REGION Network 17: PU1 Сервис
   IF #Ack OR #PU1.ack.%X3 THEN
       #errServicePU1 := FALSE;   // RS flip-flop
   END_IF;
   IF #PU1.service THEN #errServicePU1 := TRUE; END_IF;
   #PU1.st.%X3 := #errServicePU1;
END_REGION

REGION Network 18: PU2 Сервис
   IF #Ack OR #PU2.ack.%X3 THEN
       #errServicePU2 := FALSE;   // RS flip-flop
   END_IF;
   IF #PU2.service THEN #errServicePU2 := TRUE; END_IF;
   #PU2.st.%X3 := #errServicePU2;
END_REGION

REGION Network 19: Сборная ошибка РU1
   #PU1.error := #errAlarmFC_PU1 OR #errBlock_PU1 OR #errOff_KM_PU1 OR #errOn_KM_PU1 OR #errOff_UZ_PU1 OR #errON_UZ_PU1 OR #errServicePU1;
   #PU1.st.%X10 := #PU1.error;
END_REGION

REGION Network 20: Сборная ошибка РU2
   #PU2.error := #errAlarmFC_PU2 OR #errBlock_PU2 OR #errOff_KM_PU2 OR #errOn_KM_PU2 OR #errOff_UZ_PU1 OR #errON_UZ_PU1 OR #errServicePU2;
   #PU2.st.%X10 := #PU2.error;
END_REGION

REGION Network 21: Состояние работает PU1
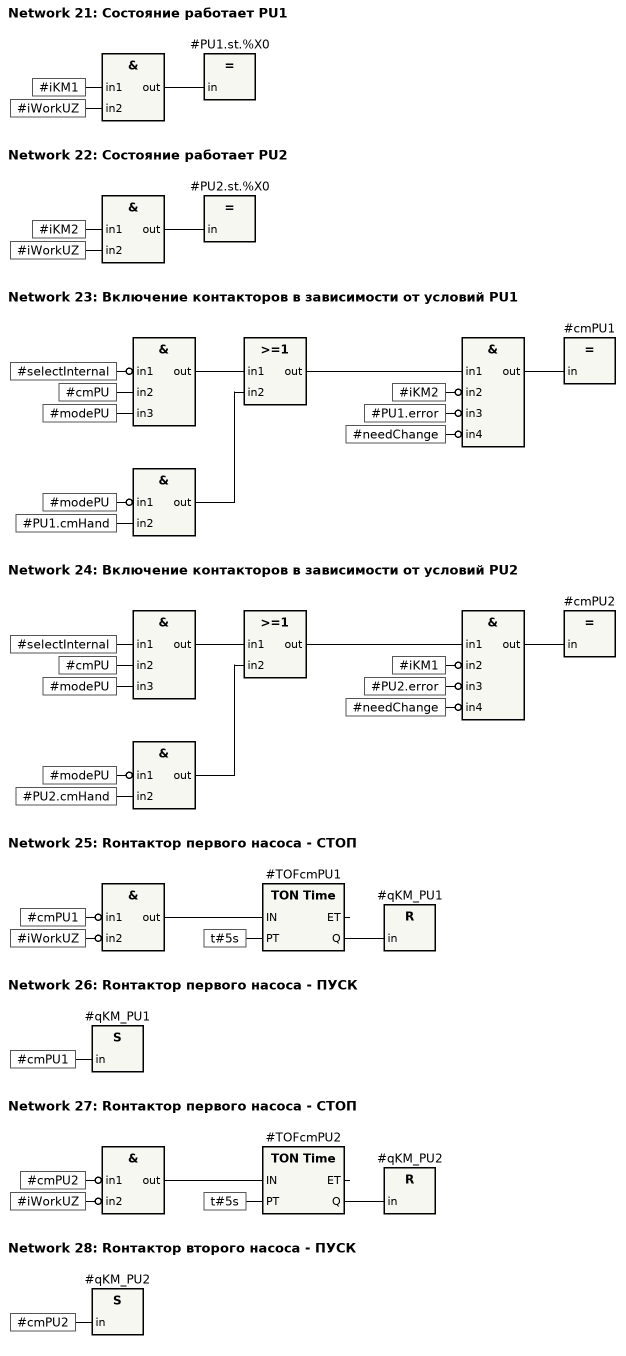
   #PU1.st.%X0 := #iKM1 AND #iWorkUZ;
END_REGION

REGION Network 22: Состояние работает PU2
   #PU2.st.%X0 := #iKM2 AND #iWorkUZ;
END_REGION

REGION Network 23: Включение контакторов в зависимости от условий PU1
   #cmPU1 := ((NOT #selectInternal AND #cmPU AND #modePU) OR (NOT #modePU AND #PU1.cmHand)) AND NOT #iKM2 AND NOT #PU1.error AND NOT #needChange;
END_REGION

REGION Network 24: Включение контакторов в зависимости от условий PU2
   #cmPU2 := ((#selectInternal AND #cmPU AND #modePU) OR (NOT #modePU AND #PU2.cmHand)) AND NOT #iKM1 AND NOT #PU2.error AND NOT #needChange;
END_REGION

REGION Network 25: Rонтактор первого насоса - СТОП
   #TOFcmPU1(IN := NOT #cmPU1 AND NOT #iWorkUZ, PT := t#5s);   // TON
   IF #TOFcmPU1.Q THEN #qKM_PU1 := FALSE; END_IF;
END_REGION

REGION Network 26: Rонтактор первого насоса - ПУСК
   IF #cmPU1 THEN #qKM_PU1 := TRUE; END_IF;
END_REGION

REGION Network 27: Rонтактор первого насоса - СТОП
   #TOFcmPU2(IN := NOT #cmPU2 AND NOT #iWorkUZ, PT := t#5s);   // TON
   IF #TOFcmPU2.Q THEN #qKM_PU2 := FALSE; END_IF;
END_REGION

REGION Network 28: Rонтактор второго насоса - ПУСК
   IF #cmPU2 THEN #qKM_PU2 := TRUE; END_IF;
END_REGION

REGION Network 29: Команда на UZ
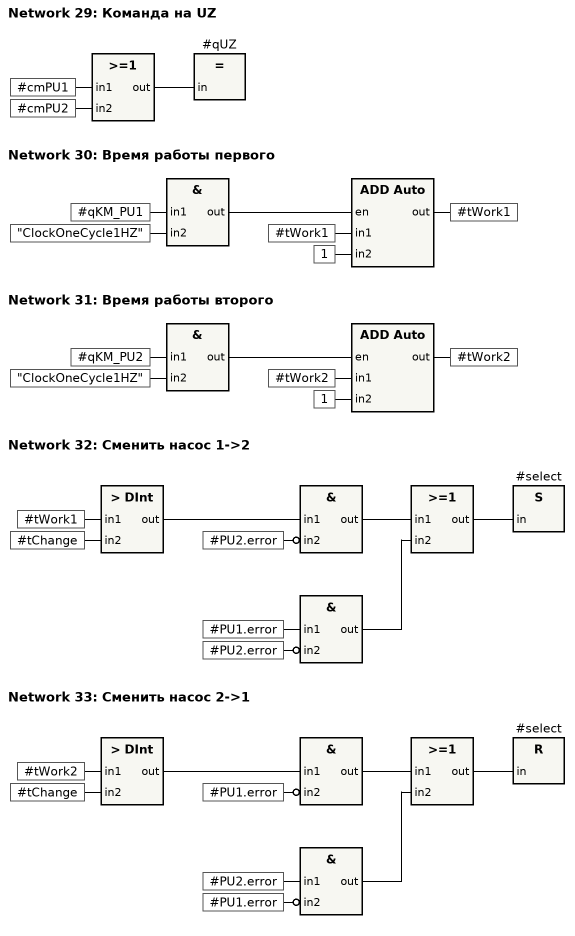
   #qUZ := #cmPU1 OR #cmPU2;
END_REGION

REGION Network 30: Время работы первого
   IF #qKM_PU1 AND "ClockOneCycle1HZ" THEN #tWork1 := #tWork1 + 1; END_IF;
END_REGION

REGION Network 31: Время работы второго
   IF #qKM_PU2 AND "ClockOneCycle1HZ" THEN #tWork2 := #tWork2 + 1; END_IF;
END_REGION

REGION Network 32: Сменить насос 1->2
   IF ((#tWork1 > #tChange) AND NOT #PU2.error) OR (#PU1.error AND NOT #PU2.error) THEN
       #select := TRUE;
   END_IF;
END_REGION

REGION Network 33: Сменить насос 2->1
   IF ((#tWork2 > #tChange) AND NOT #PU1.error) OR (#PU2.error AND NOT #PU1.error) THEN
       #select := FALSE;
   END_IF;
END_REGION

REGION Network 34
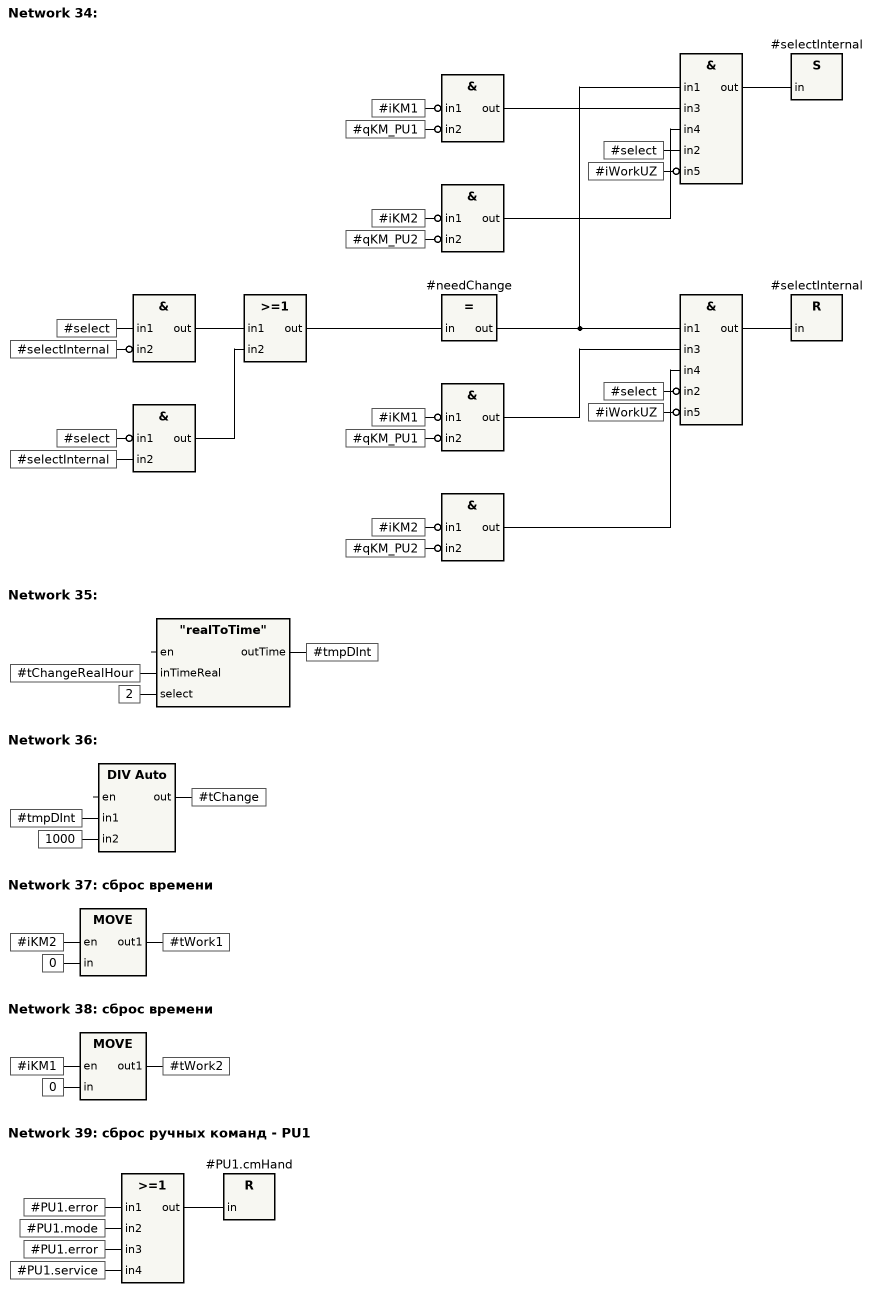
   #needChange := (#select AND NOT #selectInternal) OR (NOT #select AND #selectInternal);
   IF #needChange AND NOT #iKM1 AND NOT #qKM_PU1 AND NOT #iKM2 AND NOT #qKM_PU2 AND #select AND NOT #iWorkUZ THEN
       #selectInternal := TRUE;
   END_IF;
   IF #needChange AND NOT #iKM1 AND NOT #qKM_PU1 AND NOT #iKM2 AND NOT #qKM_PU2 AND NOT #select AND NOT #iWorkUZ THEN
       #selectInternal := FALSE;
   END_IF;
END_REGION

REGION Network 35
   "realToTime"(inTimeReal := #tChangeRealHour, select := 2, outTime => #tmpDInt);
END_REGION

REGION Network 36
   #tChange := #tmpDInt / 1000;
END_REGION

REGION Network 37: сброс времени
   IF #iKM2 THEN #tWork1 := 0; END_IF;
END_REGION

REGION Network 38: сброс времени
   IF #iKM1 THEN #tWork2 := 0; END_IF;
END_REGION

REGION Network 39: сброс ручных команд - PU1
   IF #PU1.error OR #PU1.mode OR #PU1.error OR #PU1.service THEN #PU1.cmHand := FALSE; END_IF;
END_REGION

REGION Network 40: ручная команда - PU2
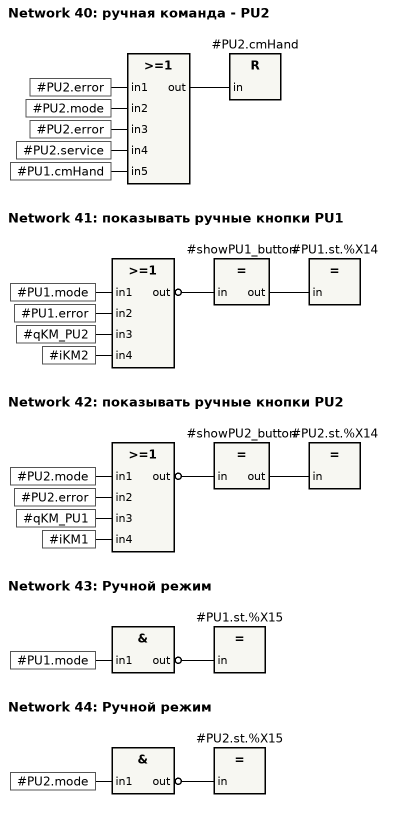
   IF #PU2.error OR #PU2.mode OR #PU2.error OR #PU2.service OR #PU1.cmHand THEN #PU2.cmHand := FALSE; END_IF;
END_REGION

REGION Network 41: показывать ручные кнопки PU1
   #showPU1_button := NOT (#PU1.mode OR #PU1.error OR #qKM_PU2 OR #iKM2);
   #PU1.st.%X14 := #showPU1_button;
END_REGION

REGION Network 42: показывать ручные кнопки PU2
   #showPU2_button := NOT (#PU2.mode OR #PU2.error OR #qKM_PU1 OR #iKM1);
   #PU2.st.%X14 := #showPU2_button;
END_REGION

REGION Network 43: Ручной режим
   #PU1.st.%X15 := NOT #PU1.mode;
END_REGION

REGION Network 44: Ручной режим
   #PU2.st.%X15 := NOT #PU2.mode;
END_REGION

REGION Network 45 (SCL): Сброс битов Ack
   IF NOT #PU1.st.%X0 AND #PU1.ack.%X0 THEN
       #PU1.ack.%X0 := 0;
   END_IF;
   IF NOT #PU1.st.%X1 AND #PU1.ack.%X1 THEN
       #PU1.ack.%X1 := 0;
   END_IF;
   IF NOT #PU1.st.%X2 AND #PU1.ack.%X2 THEN
       #PU1.ack.%X2 := 0;
   END_IF;
   IF NOT #PU1.st.%X3 AND #PU1.ack.%X3 THEN
       #PU1.ack.%X3 := 0;
   END_IF;
   IF NOT #PU1.st.%X4 AND #PU1.ack.%X4 THEN
       #PU1.ack.%X4 := 0;
   END_IF;
   IF NOT #PU1.st.%X5 AND #PU1.ack.%X5 THEN
       #PU1.ack.%X5 := 0;
   END_IF;
   IF NOT #PU1.st.%X6 AND #PU1.ack.%X6 THEN
       #PU1.ack.%X6 := 0;
   END_IF;
   IF NOT #PU1.st.%X7 AND #PU1.ack.%X7 THEN
       #PU1.ack.%X7 := 0;
   END_IF;
   IF NOT #PU1.st.%X8 AND #PU1.ack.%X8 THEN
       #PU1.ack.%X8 := 0;
   END_IF;
   IF NOT #PU1.st.%X9 AND #PU1.ack.%X9 THEN
       #PU1.ack.%X9 := 0;
   END_IF;
   IF NOT #PU1.st.%X10 AND #PU1.ack.%X10 THEN
       #PU1.ack.%X10 := 0;
   END_IF;
   IF NOT #PU1.st.%X11 AND #PU1.ack.%X11 THEN
       #PU1.ack.%X11 := 0;
   END_IF;
   IF NOT #PU1.st.%X12 AND #PU1.ack.%X12 THEN
       #PU1.ack.%X12 := 0;
   END_IF;
   IF NOT #PU1.st.%X13 AND #PU1.ack.%X13 THEN
       #PU1.ack.%X13 := 0;
   END_IF;
   IF NOT #PU1.st.%X14 AND #PU1.ack.%X14 THEN
       #PU1.ack.%X14 := 0;
   END_IF;
   IF NOT #PU1.st.%X15 AND #PU1.ack.%X15 THEN
       #PU1.ack.%X15 := 0;
   END_IF;
   IF NOT #PU2.st.%X0 AND #PU2.ack.%X0 THEN
       #PU2.ack.%X0 := 0;
   END_IF;
   IF NOT #PU2.st.%X1 AND #PU2.ack.%X1 THEN
       #PU2.ack.%X1 := 0;
   END_IF;
   IF NOT #PU2.st.%X2 AND #PU2.ack.%X2 THEN
       #PU2.ack.%X2 := 0;
   END_IF;
   IF NOT #PU2.st.%X3 AND #PU2.ack.%X3 THEN
       #PU2.ack.%X3 := 0;
   END_IF;
   IF NOT #PU2.st.%X4 AND #PU2.ack.%X4 THEN
       #PU2.ack.%X4 := 0;
   END_IF;
   IF NOT #PU2.st.%X5 AND #PU2.ack.%X5 THEN
       #PU2.ack.%X5 := 0;
   END_IF;
   IF NOT #PU2.st.%X6 AND #PU2.ack.%X6 THEN
       #PU2.ack.%X6 := 0;
   END_IF;
   IF NOT #PU2.st.%X7 AND #PU2.ack.%X7 THEN
       #PU2.ack.%X7 := 0;
   END_IF;
   IF NOT #PU2.st.%X8 AND #PU2.ack.%X8 THEN
       #PU2.ack.%X8 := 0;
   END_IF;
   IF NOT #PU2.st.%X9 AND #PU2.ack.%X9 THEN
       #PU2.ack.%X9 := 0;
   END_IF;
   IF NOT #PU2.st.%X10 AND #PU2.ack.%X10 THEN
       #PU2.ack.%X10 := 0;
   END_IF;
   IF NOT #PU2.st.%X11 AND #PU2.ack.%X11 THEN
       #PU2.ack.%X11 := 0;
   END_IF;
   IF NOT #PU2.st.%X12 AND #PU2.ack.%X12 THEN
       #PU2.ack.%X12 := 0;
   END_IF;
   IF NOT #PU2.st.%X13 AND #PU2.ack.%X13 THEN
       #PU2.ack.%X13 := 0;
   END_IF;
   IF NOT #PU2.st.%X14 AND #PU2.ack.%X14 THEN
       #PU2.ack.%X14 := 0;
   END_IF;
   IF NOT #PU2.st.%X15 AND #PU2.ack.%X15 THEN
       #PU2.ack.%X15 := 0;
   END_IF;
END_REGION
END_FUNCTION_BLOCK

FUNCTION "bitToWord" : Void   // FC5, LAD
{ S7_Optimized_Access := 'TRUE' }
VERSION : 0.1
// stored: AutoNumber true, IsIECCheckEnabled false, SetENOAutomatically false, UDAEnableTagReadback false
   VAR_INPUT
      inBit0 : Bool;
      inBit1 : Bool;
      inBit2 : Bool;
      inBit3 : Bool;
      inBit4 : Bool;
      inBit5 : Bool;
      inBit6 : Bool;
      inBit7 : Bool;
      inBit8 : Bool;
      inBit9 : Bool;
      inBit10 : Bool;
      inBit11 : Bool;
      inBit12 : Bool;
      inBit13 : Bool;
      inBit14 : Bool;
      inBit15 : Bool;
   END_VAR
   VAR_OUTPUT
      outWord : Word;
   END_VAR
BEGIN

REGION Network 1
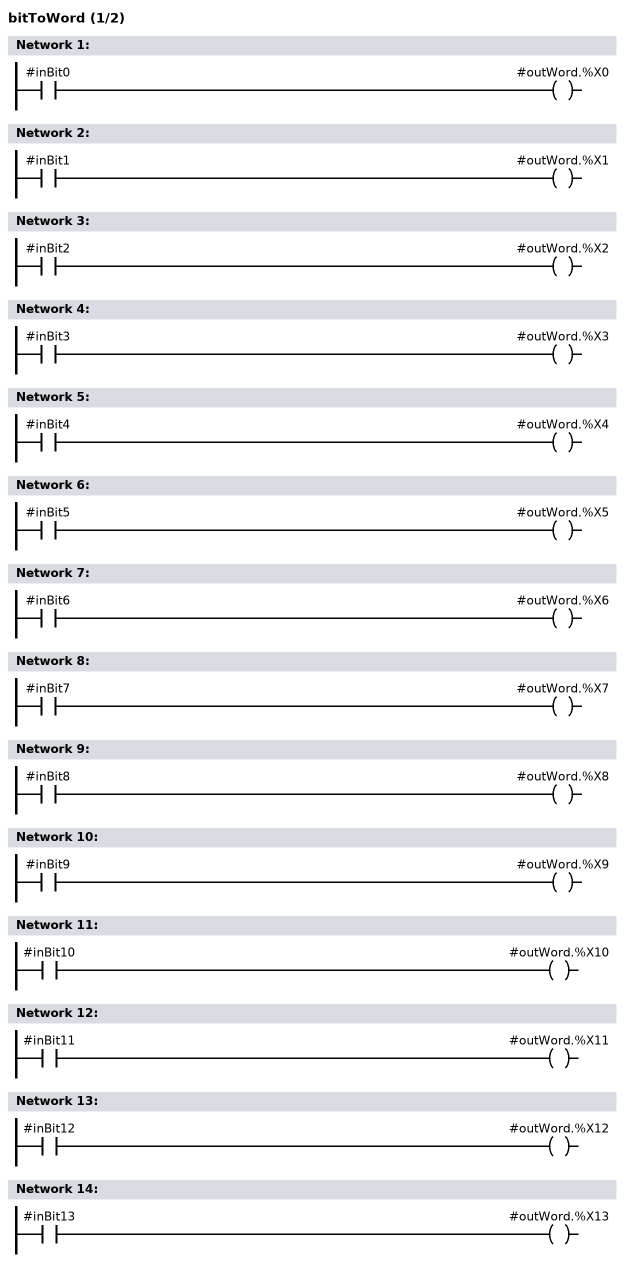
   RUNG wire#powerrail
      Contact( #inBit0 )
      Coil( #outWord.%X0 )
   END_RUNG
   // the same network as SCL:
   #outWord.%X0 := #inBit0;
END_REGION

REGION Network 2
   RUNG wire#powerrail
      Contact( #inBit1 )
      Coil( #outWord.%X1 )
   END_RUNG
   // the same network as SCL:
   #outWord.%X1 := #inBit1;
END_REGION

REGION Network 3
   RUNG wire#powerrail
      Contact( #inBit2 )
      Coil( #outWord.%X2 )
   END_RUNG
   // the same network as SCL:
   #outWord.%X2 := #inBit2;
END_REGION

REGION Network 4
   RUNG wire#powerrail
      Contact( #inBit3 )
      Coil( #outWord.%X3 )
   END_RUNG
   // the same network as SCL:
   #outWord.%X3 := #inBit3;
END_REGION

REGION Network 5
   RUNG wire#powerrail
      Contact( #inBit4 )
      Coil( #outWord.%X4 )
   END_RUNG
   // the same network as SCL:
   #outWord.%X4 := #inBit4;
END_REGION

REGION Network 6
   RUNG wire#powerrail
      Contact( #inBit5 )
      Coil( #outWord.%X5 )
   END_RUNG
   // the same network as SCL:
   #outWord.%X5 := #inBit5;
END_REGION

REGION Network 7
   RUNG wire#powerrail
      Contact( #inBit6 )
      Coil( #outWord.%X6 )
   END_RUNG
   // the same network as SCL:
   #outWord.%X6 := #inBit6;
END_REGION

REGION Network 8
   RUNG wire#powerrail
      Contact( #inBit7 )
      Coil( #outWord.%X7 )
   END_RUNG
   // the same network as SCL:
   #outWord.%X7 := #inBit7;
END_REGION

REGION Network 9
   RUNG wire#powerrail
      Contact( #inBit8 )
      Coil( #outWord.%X8 )
   END_RUNG
   // the same network as SCL:
   #outWord.%X8 := #inBit8;
END_REGION

REGION Network 10
   RUNG wire#powerrail
      Contact( #inBit9 )
      Coil( #outWord.%X9 )
   END_RUNG
   // the same network as SCL:
   #outWord.%X9 := #inBit9;
END_REGION

REGION Network 11
   RUNG wire#powerrail
      Contact( #inBit10 )
      Coil( #outWord.%X10 )
   END_RUNG
   // the same network as SCL:
   #outWord.%X10 := #inBit10;
END_REGION

REGION Network 12
   RUNG wire#powerrail
      Contact( #inBit11 )
      Coil( #outWord.%X11 )
   END_RUNG
   // the same network as SCL:
   #outWord.%X11 := #inBit11;
END_REGION

REGION Network 13
   RUNG wire#powerrail
      Contact( #inBit12 )
      Coil( #outWord.%X12 )
   END_RUNG
   // the same network as SCL:
   #outWord.%X12 := #inBit12;
END_REGION

REGION Network 14
   RUNG wire#powerrail
      Contact( #inBit13 )
      Coil( #outWord.%X13 )
   END_RUNG
   // the same network as SCL:
   #outWord.%X13 := #inBit13;
END_REGION

REGION Network 15
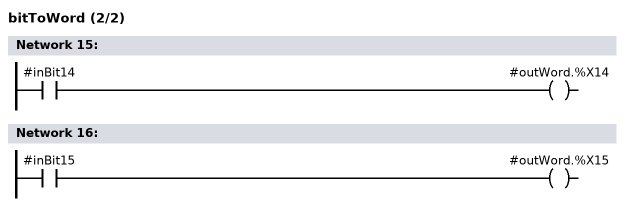
   RUNG wire#powerrail
      Contact( #inBit14 )
      Coil( #outWord.%X14 )
   END_RUNG
   // the same network as SCL:
   #outWord.%X14 := #inBit14;
END_REGION

REGION Network 16
   RUNG wire#powerrail
      Contact( #inBit15 )
      Coil( #outWord.%X15 )
   END_RUNG
   // the same network as SCL:
   #outWord.%X15 := #inBit15;
END_REGION
END_FUNCTION

FUNCTION "VLT_PROFI_FC_BASIC" : Void
TITLE = VLT_PROFI_FC_BASIC
{ S7_Optimized_Access := 'FALSE' }
AUTHOR : Danfoss_Drives
FAMILY : VLT
VERSION : 1.12
//Basic Operation Function Block
   VAR_INPUT 
      sim : Bool;
      ADR : HW_IO;   // S7-1200/1500 requires HW Identifier. Can be found in HW configuration for the specific PPO type
      DRV_EN : Bool;   // Enable Drive. Setting the Drive in Ready to Start mode.
      RUN : Bool;   // Run/Stop drive
      REVERSE : Bool;   // Drive Reverse mode. Also set P4-10 to "both directions" to allow.
      RESET : Bool;   // Reset alarms. Only Trip, not Trip lock.
      REF_VALUE : Real;   // Reference speed 0 - 10000 = 0 - 100.00%
   END_VAR

   VAR_OUTPUT 
      UZ : "UZ_Data";
   END_VAR

   VAR_TEMP 
      PCDRead : Struct   // Pointer to data structure for FC data
         STW : Struct   // Status word
            BIT_00_CTRL_RDY : Bool;   // 0=Control not ready, 1=Control ready
            BIT_01_DRV_RDY : Bool;   // 0=Frequency converter, 1=Frequency converter ready
            BIT_02_COAST_RDY : Bool;   // 0=Coasting, 1=Enable
            BIT_03_TRIP : Bool;   // 0=No error, 1=Trip
            BIT_04_ERROR : Bool;   // 0=No error, 1=Error (no trip)
            BIT_05_RESERVED : Bool;   // 0=Reserved, 1=---
            BIT_06_TRIPLOCK : Bool;   // 0=No error, 1=Triplock
            BIT_07_WARNING : Bool;   // 0=No warning, 1=Warning
            BIT_08_RUNNING_REF : Bool;   // 0=Speed <> reference, 1=Speed=reference
            BIT_09_CTRL_SOURCE : Bool;   // 0=Local operation, 1=Bus control
            BIT_10_F_LIMIT_OK : Bool;   // 0=Out of frequency limit, 1=Frequency limit ok
            BIT_11_IN_OPR : Bool;   // 0=No operation, 1=In operation
            BIT_12_IN_AUTOSTART : Bool;   // 0=Frequency converter OK, 1=Stopped, autostart
            BIT_13_VOLT_MAX : Bool;   // 0=Voltage OK, 1=Voltage exceeded
            BIT_14_TORQ_MAX : Bool;   // 0=Torque OK, 1=Torque exceeded
            BIT_15_TIMER_EXD : Bool;   // 0=Timer OK, 1=Timer exceeded
         END_STRUCT;
         MAV : Int;   // Main actual value
         PCD_02 : Int;   // PCD 02
         PCD_03 : Int;   // PCD 03
         PCD_04 : Int;   // PCD 04
         PCD_05 : Int;   // PCD 05
      END_STRUCT;
      PCDWrite : Struct   // Pointer to data structure for FC data
         CTW : Struct   // Control word
            BIT_00_PRESET_REF_1 : Bool;   // 0=Reference value, 1=selection lsb
            BIT_01_PRESET_REF_2 : Bool;   // 0=Reference value, 1=selection msb
            BIT_02_DC_BRAKE_RAMP : Bool;   // 0=DC brake, 1=Ramp
            BIT_03_COAST_INV : Bool;   // 0=Coasting, 1=No coasting
            BIT_04_QSTP_RMP : Bool;   // 0=Quick stop, 1=Ramp
            BIT_05_HLD_RMP : Bool;   // 0=Hold output frequency, 1=Use ramp
            BIT_06_START : Bool;   // 0=Ramp stop, 1=Start
            BIT_07_RESET : Bool;   // 0=No function, 1=Reset
            BIT_08_JOG : Bool;   // 0=No function, 1=Jog
            BIT_09_RAMP_1_2 : Bool;   // 0=Ramp 1, 1=Ramp 2
            BIT_10_DATA_VALID : Bool;   // 0=Dont use CTW, 1= Use CTW
            BIT_11_RLY_1_ON : Bool;   // 0=Relay 01 deactived, 1=Relay 01 active
            BIT_12_RLY_2_ON : Bool;   // 0=Relay 02 deactived, 1=Relay 02 active
            BIT_13_SETUP_SEL_1 : Bool;   // 0=Parameter set-up, 1=selection lsb
            BIT_14_SETUP_SEL_2 : Bool;   // 0=Parameter set-up, 1=selection msb
            BIT_15_REVERSE : Bool;   // 0= No Reverse, 1= Reverse
         END_STRUCT;
         MRV : Int;   // Main reference value
         PCD_02 : Int;   // PCD 02
         PCD_03 : Int;   // PCD 03
         PCD_04 : Int;   // PCD 04
         PCD_05 : Int;   // PCD 05
      END_STRUCT;
      RDRaw_Data : Array[0..5] of Int;   // Data Read. PROFINET:PPO6 only, with 4 words /PROFIBUS:PPO2 only, with 6 words
      WRRaw_Data : Array[0..5] of Int;   // Data Write. PROFINET:PPO6 only, with 4 words /PROFIBUS:PPO2 only, with 6 words
      RETVAL : Int;   // Return value for DPRD and DPWR for PNET Comm. 0=no fault
      CalcSlope : Real;   // Slope of Ref. value, to convert 0-10000 into 0- 16384
      CurrentInternal : DWord;   // Internal value for current calculation
      PowerInternal : DWord;
      AlwaysOn : Bool;   // Always on
      AlwaysOff : Bool;   // Always off
   END_VAR


BEGIN
	IF #sim THEN
	    #UZ.Ready := 1;
	    #UZ.Fault := 0;
	    #UZ.Warning := 0;
	    #UZ.ErrorConnection := 0;
	    IF #RUN THEN
	        #UZ.MAV := #REF_VALUE;
	        #UZ.Running := 1;
	    ELSE
	        #UZ.MAV := 0;
	        #UZ.Running := 0;
	    END_IF;
	    
	ELSE
	    
	    //-------------------------------------------------------------------------------------------------------------
	    // VLT_PROFI_FC_BASIC: Rev. V1.12
	    // Valid for S7-1200 and S7-1500 Type CPU's.
	    // Block handles communication with a VLT frequency converter. Either Trough PROFINET OR PROFIBUS.
	    // The FC handles basic needs and extraction of Motor current.
	    // PROFINET PPO type is PPO6 (4 words read/Write). PCD2 and PCD3 must be configured for Motor Current.
	    // PROFIBUS PPO type is PPO2 (6 words read/Write). PCD2 and PCD3 must be configured for Motor Current.
	    // Can be done in HW config of S7, on the Drive LCP or MCT10.
	    //-------------------------------------------------------------------------------------------------------------
	    
	    //------------------------------------Standard - Control bits--------------------------------------------------
	    //Can be used locally in Block.
	    #AlwaysOff := false;
	    #AlwaysOn := TRUE;
	    //------------------------------------Standard - Control bits--------------------------------------------------
	    
	    //------------------------------------Read data from fieldbus--------------------------------------------------
	    // Actual data size that is read depends on the Array size.
	    // Minimum size is 4 words.
	    // PPO type can be larger but only the 4 first words are read.
	    // Return value for DPRD and DPWR for PNET Comm. 0=No fault.
	    #RETVAL := DPRD_DAT(LADDR := #ADR, RECORD => #RDRaw_Data);  // Read Raw Data 
	    #UZ.comErr := #RETVAL;
	    //------------------------------------Read data from fieldbus--------------------------------------------------
	    
	    //------------------------------------Read Raw Data is mapped with PCDRead------------------------------------------------------
	    #PCDRead.STW.BIT_00_CTRL_RDY := #RDRaw_Data[0].%X0;
	    #PCDRead.STW.BIT_01_DRV_RDY := #RDRaw_Data[0].%X1;
	    #PCDRead.STW.BIT_02_COAST_RDY := #RDRaw_Data[0].%X2;
	    #PCDRead.STW.BIT_03_TRIP := #RDRaw_Data[0].%X3;
	    #PCDRead.STW.BIT_04_ERROR := #RDRaw_Data[0].%X4;
	    #PCDRead.STW.BIT_05_RESERVED := #RDRaw_Data[0].%X5;
	    #PCDRead.STW.BIT_06_TRIPLOCK := #RDRaw_Data[0].%X6;
	    #PCDRead.STW.BIT_07_WARNING := #RDRaw_Data[0].%X7;
	    #PCDRead.STW.BIT_08_RUNNING_REF := #RDRaw_Data[0].%X8;
	    #PCDRead.STW.BIT_09_CTRL_SOURCE := #RDRaw_Data[0].%X9;
	    #PCDRead.STW.BIT_10_F_LIMIT_OK := #RDRaw_Data[0].%X10;
	    #PCDRead.STW.BIT_11_IN_OPR := #RDRaw_Data[0].%X11;
	    #PCDRead.STW.BIT_12_IN_AUTOSTART := #RDRaw_Data[0].%X12;
	    #PCDRead.STW.BIT_13_VOLT_MAX := #RDRaw_Data[0].%X13;
	    #PCDRead.STW.BIT_14_TORQ_MAX := #RDRaw_Data[0].%X14;
	    #PCDRead.STW.BIT_15_TIMER_EXD := #RDRaw_Data[0].%X15;
	    
	    #PCDRead.MAV := #RDRaw_Data[1];
	    #PCDRead.PCD_02 := #RDRaw_Data[2];
	    #PCDRead.PCD_03 := #RDRaw_Data[3];
	    #PCDRead.PCD_04 := #RDRaw_Data[4];
	    #PCDRead.PCD_05 := #RDRaw_Data[5];
	    //------------------------------------Read Raw Data is mapped with PCDRead------------------------------------------------------
	    
	    //------------------------------------Extraction of Main actual value--------------------------------------------
	    // Main Actual Value(MAV) is read from the Drive as 0 - 16384. Must be converted into 0 - 10000 (0.0 - 100.0 %)
	    IF #UZ.comErr = 0 THEN
	        #CalcSlope := LREAL_TO_REAL(10000.0 / 16384.0);
	        #UZ.MAV := INT_TO_REAL(#PCDRead.MAV) / 163.84; // Convert to percentage (0.0 - 100.0)
	    END_IF;
	    //------------------------------------Extraction of Main actual value--------------------------------------------
	    
	    //------------------------------------Calculation of motor current----------------------------------------------
	    // Motor current is a 32 bit value hence 2 words read from the Drive need to be combined into a DWORD.
	    // Motor current is scaled with 2 decimal points (conversion index -2) hence division by 100.
	    IF #UZ.comErr = 0 THEN
	        #CurrentInternal := DINT_TO_DWORD(#PCDRead.PCD_02); // PCD02 is high word of Motor current
	        #CurrentInternal := SHL_DWORD(IN := #CurrentInternal, N := 16); // Shift high word of Motor current 16 bits to the left
	        #CurrentInternal := #CurrentInternal + DINT_TO_DWORD(#PCDRead.PCD_03); // PCD03 is low word of Motor current
	        #UZ.MotorCurrent := DINT_TO_REAL(DWORD_TO_DINT(#CurrentInternal)) / 100.0;
	        
	        #PowerInternal := DINT_TO_DWORD(#PCDRead.PCD_04);
	        #PowerInternal := SHL_DWORD(IN := #PowerInternal, N := 16);
	        #PowerInternal := #PowerInternal + DINT_TO_DWORD(#PCDRead.PCD_05);
	        #UZ.MotorPower := DINT_TO_REAL(DWORD_TO_DINT(#PowerInternal)) / 100.0;
	    END_IF;
	    //------------------------------------Calculation of Motor current----------------------------------------------
	    
	    //------------------------------------Mask out Drive status bit's-----------------------------------------------
	    IF #UZ.comErr = 0 THEN
	        #UZ.Ready := (#PCDRead.STW.BIT_00_CTRL_RDY AND #PCDRead.STW.BIT_01_DRV_RDY AND #PCDRead.STW.BIT_02_COAST_RDY AND #PCDRead.STW.BIT_09_CTRL_SOURCE); // Drive ready to start from Fieldbus
	        #UZ.Running := #PCDRead.STW.BIT_11_IN_OPR; // Drive is started but not necessarily running on reference speed.
	        #UZ.Run_On_ref := #PCDRead.STW.BIT_08_RUNNING_REF; // Running on reference
	        #UZ.Warning := #PCDRead.STW.BIT_07_WARNING; // Warning present
	        #UZ.Fault := (#PCDRead.STW.BIT_04_ERROR OR #PCDRead.STW.BIT_03_TRIP OR #PCDRead.STW.BIT_06_TRIPLOCK); // Fault present. Trip or Trip lock
	    ELSE
	        #UZ.Ready := FALSE;
	        #UZ.Fault := TRUE;
	    END_IF;
	    //------------------------------------Mask out Drive status bit's-----------------------------------------------
	    
	    //------------------------------------Default settings of Controlword-------------------------------------------
	    // Prepare all Controlword Bit's to default values so that
	    // they are in a "ready to start" mode. CTW =043Ch
	    #PCDWrite.CTW.BIT_00_PRESET_REF_1 := FALSE;
	    #PCDWrite.CTW.BIT_01_PRESET_REF_2 := FALSE;
	    
	    IF #DRV_EN THEN
	        #PCDWrite.CTW.BIT_02_DC_BRAKE_RAMP := TRUE;
	        #PCDWrite.CTW.BIT_03_COAST_INV := TRUE;
	        #PCDWrite.CTW.BIT_04_QSTP_RMP := TRUE;
	        #PCDWrite.CTW.BIT_05_HLD_RMP := TRUE;
	    ELSE
	        #PCDWrite.CTW.BIT_02_DC_BRAKE_RAMP := FALSE;
	        #PCDWrite.CTW.BIT_03_COAST_INV := FALSE;
	        #PCDWrite.CTW.BIT_04_QSTP_RMP := FALSE;
	        #PCDWrite.CTW.BIT_05_HLD_RMP := FALSE;
	    END_IF;
	    
	    #PCDWrite.CTW.BIT_06_START := FALSE;
	    #PCDWrite.CTW.BIT_07_RESET := FALSE;
	    #PCDWrite.CTW.BIT_08_JOG := FALSE;
	    #PCDWrite.CTW.BIT_09_RAMP_1_2 := FALSE;
	    #PCDWrite.CTW.BIT_10_DATA_VALID := TRUE;
	    #PCDWrite.CTW.BIT_11_RLY_1_ON := FALSE;
	    #PCDWrite.CTW.BIT_12_RLY_2_ON := FALSE;
	    #PCDWrite.CTW.BIT_13_SETUP_SEL_1 := FALSE;
	    #PCDWrite.CTW.BIT_14_SETUP_SEL_2 := FALSE;
	    #PCDWrite.CTW.BIT_15_REVERSE := FALSE;
	    //------------------------------------Default settings of Controlword-------------------------------------------
	    
	    //------------------------------------Drive control bit's-------------------------------------------------------
	    #PCDWrite.CTW.BIT_06_START := #RUN AND NOT #UZ.Fault; // Start the Drive if there is no pending Fault.
	    #PCDWrite.CTW.BIT_15_REVERSE := #REVERSE; // Set Drive to Reverse Mode. Ensure Par. 4-10 is set to "Both Directions"
	    #PCDWrite.CTW.BIT_07_RESET := #RESET; // Reset pending Fault
	    //------------------------------------Drive control bit's-------------------------------------------------------
	    
	    //------------------------------------Reference value limit check------------------------------------------------
	    // Must be between 0 - 10000. Ensure reference speed is within limits.
	    IF #REF_VALUE >= 100.00 THEN
	        #REF_VALUE := (100.00);
	    END_IF;
	    IF #REF_VALUE < 0.0 THEN
	        #REF_VALUE := 0.0;
	    END_IF;
	    //------------------------------------Reference value limit check------------------------------------------------
	    
	    //------------------------------------PCDWrite is mapped with WriteRaw data--------------------------------------------------
	    #WRRaw_Data[0].%X0 := #PCDWrite.CTW.BIT_00_PRESET_REF_1;
	    #WRRaw_Data[0].%X1 := #PCDWrite.CTW.BIT_01_PRESET_REF_2;
	    #WRRaw_Data[0].%X2 := #PCDWrite.CTW.BIT_02_DC_BRAKE_RAMP;
	    #WRRaw_Data[0].%X3 := #PCDWrite.CTW.BIT_03_COAST_INV;
	    #WRRaw_Data[0].%X4 := #PCDWrite.CTW.BIT_04_QSTP_RMP;
	    #WRRaw_Data[0].%X5 := #PCDWrite.CTW.BIT_05_HLD_RMP;
	    #WRRaw_Data[0].%X6 := #PCDWrite.CTW.BIT_06_START;
	    #WRRaw_Data[0].%X7 := #PCDWrite.CTW.BIT_07_RESET;
	    #WRRaw_Data[0].%X8 := #PCDWrite.CTW.BIT_08_JOG;
	    #WRRaw_Data[0].%X9 := #PCDWrite.CTW.BIT_09_RAMP_1_2;
	    #WRRaw_Data[0].%X10 := #PCDWrite.CTW.BIT_10_DATA_VALID;
	    #WRRaw_Data[0].%X11 := #PCDWrite.CTW.BIT_11_RLY_1_ON;
	    #WRRaw_Data[0].%X12 := #PCDWrite.CTW.BIT_12_RLY_2_ON;
	    #WRRaw_Data[0].%X13 := #PCDWrite.CTW.BIT_13_SETUP_SEL_1;
	    #WRRaw_Data[0].%X14 := #PCDWrite.CTW.BIT_14_SETUP_SEL_2;
	    #WRRaw_Data[0].%X15 := #PCDWrite.CTW.BIT_15_REVERSE;
	    
	    #WRRaw_Data[2] := #PCDWrite.PCD_02;
	    #WRRaw_Data[3] := #PCDWrite.PCD_03;
	    //------------------------------------PCDWrite is mapped with WriteRaw data--------------------------------------------------
	    
	    //------------------------------------Reference value limit check------------------------------------------------
	    // Must be between 0 - 10000. Ensure reference speed is within limits.
	    IF #REF_VALUE >= 100.00 THEN
	        #REF_VALUE := 100.00;
	    END_IF;
	    IF #REF_VALUE < 0.0 THEN
	        #REF_VALUE := 0.0;
	    END_IF;
	    //------------------------------------Reference value limit check------------------------------------------------
	    
	    //------------------------------------Prepare Reference value----------------------------------------------------
	    // PCD Write block position 1. Fit's with PPO type mapping
	    // Convert 10000 into 16384 which equals 4000h. 10000 = 100.00%
	    #CalcSlope := LREAL_TO_REAL(16384.0 / 10000.0);
	    #PCDWrite.MRV := REAL_TO_INT(#REF_VALUE * 163.84);
	    //FLOOR_INT(#CalcSlope * #REF_VALUE); // Convert to percentage (0.0 - 100.0)
	    #WRRaw_Data[1] := #PCDWrite.MRV; // Main reference value is Mapped with write Raw Data
	    //------------------------------------Prepare Reference value----------------------------------------------------
	    
	    //------ADR------------------------------Send Data------------------------------------------------------------------
	    // Return value for DPRD and DPWR for PNET Comm. 0=No fault
	    IF #UZ.comErr = 0 THEN
	        #RETVAL := DPWR_DAT(LADDR := #ADR, RECORD := #WRRaw_Data); //#Write Raw Data);
	        #UZ.comErr := #RETVAL;
	    END_IF;
	    //------------------------------------Send Data------------------------------------------------------------------
	    
	    
	    IF #UZ.comErr = 0 THEN
	        #UZ.ErrorConnection := 0;
	    ELSE
	        #UZ.ErrorConnection := 1;
	    END_IF;
	    
	END_IF;
	
	//------------------------------------Ensure ENO is TRUE always--------------------------------------------------
	ENO := TRUE;
	//------------------------------------Ensure ENO is TRUE always--------------------------------------------------
	
END_FUNCTION

FUNCTION_BLOCK "AllDpump"
{ S7_Optimized_Access := 'TRUE' }
VERSION : 0.1
   VAR 
      dp101 : "DPumpCntr";
      dp501 : "DPumpCntr";
      dp502 : "DPumpCntr";
      dp801 : "DPumpCntr";
      dp802 : "DPumpCntr";
      dp803 : "DPumpCntr";
      dp1001 : "DPumpCntr";
   END_VAR


BEGIN
	
	REGION Dpumps handlers
	    #dp101(power := TRUE,
	           run := "iDP101_Run",
	           emrStop := TRUE,
	           alarmFC := "iDP101_Fail",
	           Ack := "dbMain".Ack,
	           FE := 0.0,
	           qStart => "qDP101_Start",
	           pqw => "aqDP101",
	           dev := "dtDpump".dp101,
	           prop := "dtPropDpump".dp101);
	    
	    #dp501(power := TRUE,
	           run := "iDP501_Run",
	           emrStop := TRUE,
	           alarmFC := "iDP501_Fail",
	           Ack := "dbMain".Ack,
	           FE := 0.0,
	           qStart => "qDP501_Start",
	           pqw => "aqDP501",
	           dev := "dtDpump".dp501,
	           prop := "dtPropDpump".dp501);
	    
	    #dp502(power := TRUE,
	           run := "iDP502_Run",
	           emrStop := TRUE,
	           alarmFC := "iDP502_Fail",
	           Ack := "dbMain".Ack,
	           FE := 0.0,
	           qStart => "qDP502_Start",
	           pqw => "aqDP502",
	           dev := "dtDpump".dp502,
	           prop := "dtPropDpump".dp502);
	    
	    #dp801(power := TRUE,
	           run := "iDP801_Run",
	           emrStop := TRUE,
	           alarmFC := "iDP801_Fail",
	           Ack := "dbMain".Ack,
	           FE := 0.0,
	           qStart => "qDP801_Start",
	           pqw => "aqDP801",
	           dev := "dtDpump".dp801,
	           prop := "dtPropDpump".dp801);
	    
	    #dp802(power := TRUE,
	           run := "iDP802_Run",
	           emrStop := TRUE,
	           alarmFC := "iDP802_Fail",
	           Ack := "dbMain".Ack,
	           FE := 0.0,
	           qStart => "qDP802_Start",
	           pqw => "aqDP802",
	           dev := "dtDpump".dp802,
	           prop := "dtPropDpump".dp802);
	    
	    #dp803(power := TRUE,
	           run := "iDP803_Run",
	           emrStop := TRUE,
	           alarmFC := "iDP803_Fail",
	           Ack := "dbMain".Ack,
	           FE := 0.0,
	           qStart => "qDP803_Start",
	           pqw => "aqDP803",
	           dev := "dtDpump".dp803,
	           prop := "dtPropDpump".dp803);
	    
	    #dp1001(power := TRUE,
	            run := "iDP1001_Run",
	            emrStop := TRUE,
	            alarmFC := "iDP1001_Fail",
	            Ack := "dbMain".Ack,
	            FE := 0.0,
	            qStart => "qDP1001_Start",
	            pqw => "aqDP1001",
	            dev := "dtDpump".dp1001,
	            prop := "dtPropDpump".dp1001);
	END_REGION
	
END_FUNCTION_BLOCK

FUNCTION_BLOCK "DPumpCntr"   // FB70, LAD
{ S7_Optimized_Access := 'FALSE' }
VERSION : 0.1
// #ST:
// номер бита, часло десятичное
//  0  - стоп 
// 0 1 - работа
// 1 2 - запуск
// 2 4 - остановка
// 3 8 - сервисный режим
// 4 16 - ошибка Пуска
// 5 32 - ошибка Стопа
// 6 64 - ошибка питания
// 7 128 - ошибка частотника (дозатора)
// 8 256 - Блокировка внешняя
// 9 - 512 - нажат аварийный стоп
// 10 -1024 - сборная авария
// 11 2048
// 12 4096
// 13 8192
// 14 16384 
// 15 32768 - режим 0-ручной, 1-авто
// 
// 
// 
// показывать кнопки ручного управления
// stored: AutoNumber false, IsIECCheckEnabled false, SetENOAutomatically false, UDAEnableTagReadback false
   VAR_INPUT
      power : Bool;   // питание устройства
      run : Bool;
      emrStop : Bool;   // Авариный стоп 0-авария, 1-ок
      alarmFC : Bool;   // 1-авария
      Ack : Bool;   // Сброс Аварий
      FE : Real;
   END_VAR
   VAR_OUTPUT
      qStart : Bool;
      pqw : Int;
   END_VAR
   VAR_IN_OUT
      dev : "DPump";
      prop : "PropDosing";
   END_VAR
   VAR DB_SPECIFIC
      ErrOC : Bool;   // Признак аварии по закрытию или открытию
      ErrPower : Bool;   // Признак аварии питания
      ErrDis : Bool;   // Признак внешней блокировки
      qON : Bool;   // Выход для управления механизмом
      tmrClosing { S7_SetPoint := 'True'} : TON_TIME;
      tmrOpening { S7_SetPoint := 'True'} : TON_TIME;
      closed : Bool;
      opened : Bool;
      closing : Bool;
      opening : Bool;
      errStart : Bool;
      errStop : Bool;
      errEmrStop : Bool;
      errAlarmFc : Bool;
      errService : Bool;
      tStart : Time;
      tStop : Time;
   END_VAR
   VAR
      ServiceEventHandler { S7_SetPoint := 'True'} : "DevAckSingleAlarm";
      PowerEventHandler { S7_SetPoint := 'True'} : "DevAckSingleAlarm";
      DevAlarmEventHandler { S7_SetPoint := 'True'} : "DevAckSingleAlarm";
      DisEventHandler { S7_SetPoint := 'True'} : "DevAckSingleAlarm";
      EmrStopEventHandler { S7_SetPoint := 'True'} : "DevAckSingleAlarm";
      BadStartEventHandler { S7_SetPoint := 'True'} : "DevAckSingleAlarm";
      BadStopEventHandler { S7_SetPoint := 'True'} : "DevAckSingleAlarm";
   END_VAR
BEGIN

REGION Network 1: Сброс состояния
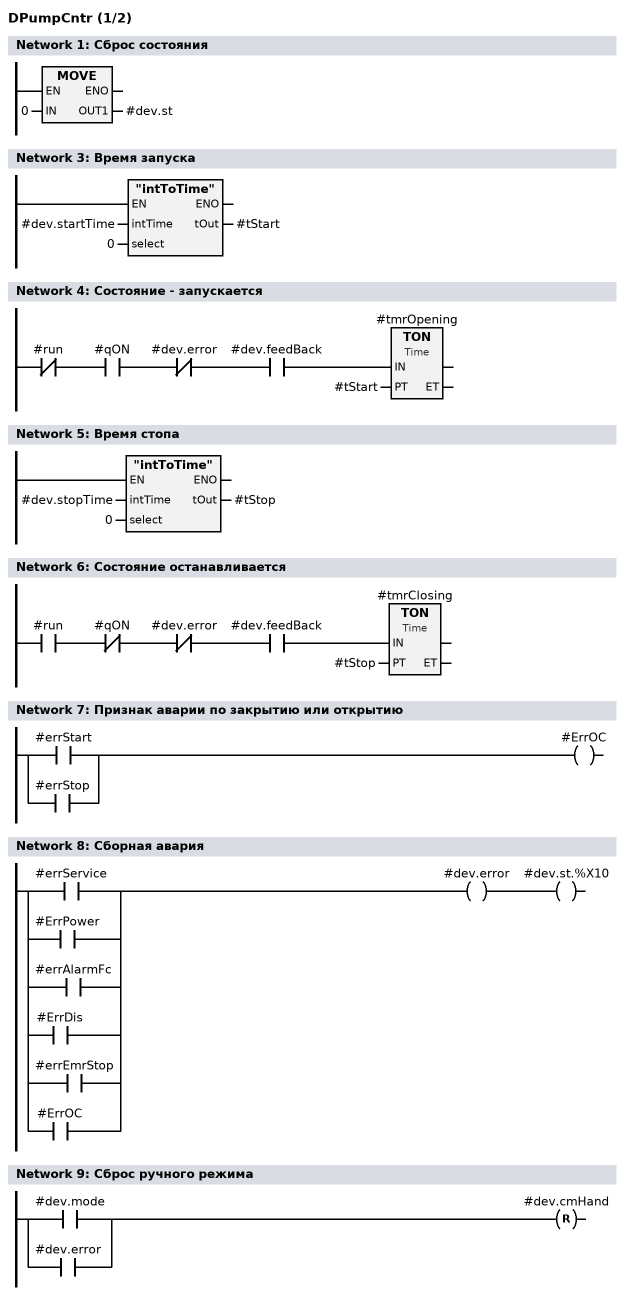
   RUNG wire#powerrail
      { S7_GenerateENO := "TRUE" } Move(in := 0, out1 => #dev.st)
   END_RUNG
   // the same network as SCL:
   #dev.st := 0;
END_REGION

REGION Network 2 (SCL): Event handlers
   #ServiceEventHandler(alarmSignal := #dev.service,
                        ack := #Ack,
                        ackBit := #dev.ack.%X3,
                        stateBit := #dev.st.%X3,
                        alarmTag := #errService);
   #BadStartEventHandler(alarmSignal:=#tmrOpening.Q,
                         ack:=#Ack,
                         ackBit:=#dev.ack.%X4,
                         stateBit:=#dev.st.%X4,
                         alarmTag:=#errStart);
   #BadStopEventHandler(alarmSignal:=#tmrClosing.Q,
                        ack:=#Ack,
                        ackBit:=#dev.ack.%X5,
                        stateBit:=#dev.ack.%X5,
                        alarmTag:=#errStop);
   #PowerEventHandler(alarmSignal := #power,
                      ack := #Ack,
                      ackBit := #dev.ack.%X6,
                      stateBit := #dev.st.%X6,
                      alarmTag := #ErrPower);
   #DevAlarmEventHandler(alarmSignal := #alarmFC,
                         ack := #Ack,
                         ackBit := #dev.ack.%X7,
                         stateBit := #dev.st.%X7,
                         alarmTag := #errAlarmFc);
   #DisEventHandler(alarmSignal := #dev.block,
                    ack := #Ack,
                    ackBit := #dev.ack.%X8,
                    stateBit := #dev.st.%X8,
                    alarmTag := #ErrDis);
   #EmrStopEventHandler(alarmSignal := #emrStop,
                        ack := #Ack,
                        ackBit := #dev.ack.%X9,
                        stateBit := #dev.st.%X9,
                        alarmTag := #errEmrStop);
END_REGION

REGION Network 3: Время запуска
   RUNG wire#powerrail
      "intToTime"(intTime := #dev.startTime, select := 0, tOut => #tStart)
   END_RUNG
   // the same network as SCL:
   "intToTime"(intTime := #dev.startTime, select := 0, tOut => #tStart);
END_REGION

REGION Network 4: Состояние - запускается
   RUNG wire#powerrail
      I_Contact( #run )
      Contact( #qON )
      I_Contact( #dev.error )
      Contact( #dev.feedBack )
      { S7_Templates := "time_type := Time" } #tmrOpening.TON(pt := #tStart, et =>)
   END_RUNG
   // the same network as SCL:
   #tmrOpening(IN := NOT #run AND #qON AND NOT #dev.error AND #dev.feedBack, PT := #tStart);   // TON
END_REGION

REGION Network 5: Время стопа
   RUNG wire#powerrail
      "intToTime"(intTime := #dev.stopTime, select := 0, tOut => #tStop)
   END_RUNG
   // the same network as SCL:
   "intToTime"(intTime := #dev.stopTime, select := 0, tOut => #tStop);
END_REGION

REGION Network 6: Состояние останавливается
   RUNG wire#powerrail
      Contact( #run )
      I_Contact( #qON )
      I_Contact( #dev.error )
      Contact( #dev.feedBack )
      { S7_Templates := "time_type := Time" } #tmrClosing.TON(pt := #tStop, et =>)
   END_RUNG
   // the same network as SCL:
   #tmrClosing(IN := #run AND NOT #qON AND NOT #dev.error AND #dev.feedBack, PT := #tStop);   // TON
END_REGION

REGION Network 7: Признак аварии по закрытию или открытию
   RUNG wire#powerrail
      Contact( #errStart )
      wire#w1
      Coil( #ErrOC )
   END_RUNG
   RUNG wire#powerrail
      Contact( #errStop )
   END_RUNG wire#w1
   // the same network as SCL:
   #ErrOC := #errStart OR #errStop;
END_REGION

REGION Network 8: Сборная авария
   RUNG wire#powerrail
      Contact( #errService )
      wire#w1
      Coil( #dev.error )
      Coil( #dev.st.%X10 )
   END_RUNG
   RUNG wire#powerrail
      Contact( #ErrPower )
   END_RUNG wire#w1
   RUNG wire#powerrail
      Contact( #errAlarmFc )
   END_RUNG wire#w1
   RUNG wire#powerrail
      Contact( #ErrDis )
   END_RUNG wire#w1
   RUNG wire#powerrail
      Contact( #errEmrStop )
   END_RUNG wire#w1
   RUNG wire#powerrail
      Contact( #ErrOC )
   END_RUNG wire#w1
   // the same network as SCL:
   #dev.error := #errService OR #ErrPower OR #errAlarmFc OR #ErrDis OR #errEmrStop OR #ErrOC;
   #dev.st.%X10 := #dev.error;
END_REGION

REGION Network 9: Сброс ручного режима
   RUNG wire#powerrail
      Contact( #dev.mode )
      wire#w1
      R_Coil( #dev.cmHand )
   END_RUNG
   RUNG wire#powerrail
      Contact( #dev.error )
   END_RUNG wire#w1
   // the same network as SCL:
   IF #dev.mode OR #dev.error THEN #dev.cmHand := FALSE; END_IF;
END_REGION

REGION Network 10: Сброс авто режима
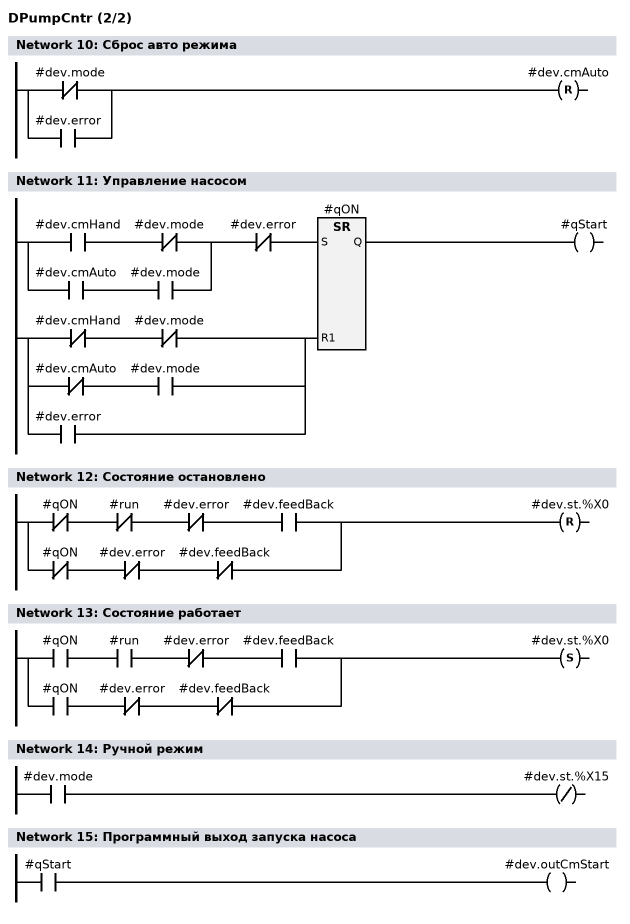
   RUNG wire#powerrail
      I_Contact( #dev.mode )
      wire#w1
      R_Coil( #dev.cmAuto )
   END_RUNG
   RUNG wire#powerrail
      Contact( #dev.error )
   END_RUNG wire#w1
   // the same network as SCL:
   IF NOT #dev.mode OR #dev.error THEN #dev.cmAuto := FALSE; END_IF;
END_REGION

REGION Network 11: Управление насосом
   RUNG wire#powerrail
      Contact( #dev.cmHand )
      I_Contact( #dev.mode )
      wire#w1
      I_Contact( #dev.error )
      S_SR(operand := #qON, r1 := wire#w2)
      Coil( #qStart )
   END_RUNG
   RUNG wire#powerrail
      Contact( #dev.cmAuto )
      Contact( #dev.mode )
   END_RUNG wire#w1
   RUNG wire#powerrail
      I_Contact( #dev.cmHand )
      I_Contact( #dev.mode )
   END_RUNG wire#w2
   RUNG wire#powerrail
      I_Contact( #dev.cmAuto )
      Contact( #dev.mode )
   END_RUNG wire#w2
   RUNG wire#powerrail
      Contact( #dev.error )
   END_RUNG wire#w2
   // the same network as SCL:
   IF ((#dev.cmHand AND NOT #dev.mode) OR (#dev.cmAuto AND #dev.mode)) AND NOT #dev.error THEN
       #qON := TRUE;   // SR flip-flop
   END_IF;
   IF (NOT #dev.cmHand AND NOT #dev.mode) OR (NOT #dev.cmAuto AND #dev.mode) OR #dev.error THEN
       #qON := FALSE;
   END_IF;
   #qStart := #qON;
END_REGION

REGION Network 12: Состояние остановлено
   RUNG wire#powerrail
      I_Contact( #qON )
      I_Contact( #run )
      I_Contact( #dev.error )
      Contact( #dev.feedBack )
      wire#w1
      R_Coil( #dev.st.%X0 )
   END_RUNG
   RUNG wire#powerrail
      I_Contact( #qON )
      I_Contact( #dev.error )
      I_Contact( #dev.feedBack )
   END_RUNG wire#w1
   // the same network as SCL:
   IF (NOT #qON AND NOT #run AND NOT #dev.error AND #dev.feedBack) OR (NOT #qON AND NOT #dev.error AND NOT #dev.feedBack) THEN
       #dev.st.%X0 := FALSE;
   END_IF;
END_REGION

REGION Network 13: Состояние работает
   RUNG wire#powerrail
      Contact( #qON )
      Contact( #run )
      I_Contact( #dev.error )
      Contact( #dev.feedBack )
      wire#w1
      S_Coil( #dev.st.%X0 )
   END_RUNG
   RUNG wire#powerrail
      Contact( #qON )
      I_Contact( #dev.error )
      I_Contact( #dev.feedBack )
   END_RUNG wire#w1
   // the same network as SCL:
   IF (#qON AND #run AND NOT #dev.error AND #dev.feedBack) OR (#qON AND NOT #dev.error AND NOT #dev.feedBack) THEN
       #dev.st.%X0 := TRUE;
   END_IF;
END_REGION

REGION Network 14: Ручной режим
   RUNG wire#powerrail
      Contact( #dev.mode )
      I_Coil( #dev.st.%X15 )
   END_RUNG
   // the same network as SCL:
   #dev.st.%X15 := NOT #dev.mode;
END_REGION

REGION Network 15: Программный выход запуска насоса
   RUNG wire#powerrail
      Contact( #qStart )
      Coil( #dev.outCmStart )
   END_RUNG
   // the same network as SCL:
   #dev.outCmStart := #qStart;
END_REGION

REGION Network 16 (SCL): Prop dossing
   //дозирование пропорционально расходу

   //производителньность л/ч

   IF #dev.mode AND #dev.cmAuto THEN
       //KVA
       IF #prop.enableFix THEN
           IF #prop.fixSP > 100 THEN
               #prop.fixSP := 100;
           END_IF;
           IF #prop.fixSP < 0 THEN
               #prop.fixSP := 0;
           END_IF;
           #prop.outLPH := (#prop.max * #prop.fixSP) / 100;
           //
           // #prop.outLPH := #prop.fixSP;
       ELSE
           IF #prop.density > 0 THEN
               #prop.outLPH := #FE * #prop.spAuto / (#prop.density * 1000.0);
           ELSE
               #prop.outLPH := 0;
           END_IF;

           //запрет дозирования если расход меньше заданного
           IF #FE < #prop.minFE THEN
               #prop.outLPH := 0.0;
           END_IF;
       END_IF;
   END_IF;
   IF NOT #dev.mode AND #dev.cmHand THEN
       #prop.outLPH := #prop.spHand;
   END_IF;

   //запрет дозирования
   IF NOT #dev.cmHand AND NOT #dev.cmAuto THEN
       #prop.outLPH := 0.0;
   END_IF;

   IF #prop.outLPH > #prop.max THEN
       #prop.outLPH := #prop.max;
   END_IF;

   //расчет PQW
   IF #prop.max > 0 THEN
       #pqw := REAL_TO_INT(#prop.outLPH * 27648.0 / #prop.max);
   ELSE
       #pqw := 0;
   END_IF;

   //ограничение выхода
   IF #pqw < 0 THEN
       #pqw := 0;
   END_IF;
   IF #pqw > 27648 THEN
       #pqw := 27648;
   END_IF;
   //расчет тока
   #prop.outmA := 4.0 + INT_TO_REAL(#pqw) * 16.0 / 27648.0;
   #prop.outSP := INT_TO_REAL(#pqw) * 100.0 / 27648.0;
   #prop.FE := #FE;
END_REGION
END_FUNCTION_BLOCK

FUNCTION_BLOCK "AllUF"
{ S7_Optimized_Access := 'TRUE' }
VERSION : 0.1
   VAR 
      reqNumbWorkUF { ExternalVisible := 'False'; ExternalWritable := 'False'} : USInt;
      readyUF : Array[0..1] of Bool;
      workUF : Array[0..1] of Bool;
      cmUF : Array[0..1] of Bool;
      HandlerUF1 : "HandlerUF";
      HandlerUF2 : "HandlerUF";
   END_VAR

   VAR_TEMP 
      tChModeUF1 : Bool;
      tChModeUF2 : Bool;
      tErr : Bool;
   END_VAR

   VAR CONSTANT 
      UF1 : Int := 0;
      UF2 : Int := 1;
   END_VAR


BEGIN
	REGION Device mode for UF12 and UF34
	    //Valves UF1
	    "dtAV".DVA501.mode :=
	    "dtAV".DVA503.mode :=
	    "dtAV".DVA505.mode :=
	    "dtAV".DVA507.mode :=
	    "dtAV".DVA508.mode :=
	    "dtAV".DVA509.mode :=
	    "dtAV".DVA512.mode :=
	    "dtUF".modeUF1;
	    //Valves UF2
	    "dtAV".DVA502.mode :=
	    "dtAV".DVA510.mode :=
	    "dtAV".DVA513.mode :=
	    "dtAV".DVA514.mode :=
	    "dtAV".DVA515.mode :=
	    "dtAV".DVA516.mode :=
	    "dtAV".DVA506.mode :=
	    "dtUF".modeUF2;
	    //Common devices
	    "dtAV".DVA504.mode :=
	    "dtAV".DVA511.mode :=
	    //    "dtPump".P701.mode :=
	    //    "dtPump".P701.mode :=
	    "dtUF".modeUF1 OR "dtUF".modeUF2;
	END_REGION
	REGION Calculate number of UF in work
	    // "CalcNumDevUf"(cmStart:= "dtUF".cmAuto,
	    //                nWorkDev:=#reqNumbWorkUF,
	    //                lev:= "dtAnalogData".et_data["aiLT601"].Par,
	    //                levStop1:="dtParmUF".filtrateStopLevUF1,
	    //                levStart1:="dtParmUF".filtrateStartLevUF1,
	    //                levStop2:="dtParmUF".filtrateStopLevUF2,
	    //                levStart2:="dtParmUF".filtrateStartLevUF2,
	    //                settingsError=>"dtParmUF".errSettingsLev,
	    //                nNeedWork:=#reqNumbWorkUF);
	END_REGION
	REGION Prepare FOR select work UF
	    #readyUF[#UF1] := "dtUF".modeUF1
	    AND NOT (
	    "dtUF".flagUF1.Err OR
	    "dtUF".flagUF1.HW OR
	    "dtUF".flagUF1.HW_A OR
	    "dtUF".flagUF1.CEB1 OR
	    "dtUF".flagUF1.CEB1_A OR
	    "dtUF".flagUF1.CEB2 OR
	    "dtUF".flagUF1.CEB2_A
	    );
	    #readyUF[#UF2] := "dtUF".modeUF2
	    AND NOT (
	    "dtUF".flagUF2.Err OR
	    "dtUF".flagUF2.HW OR
	    "dtUF".flagUF2.HW_A OR
	    "dtUF".flagUF2.CEB1 OR
	    "dtUF".flagUF2.CEB1_A OR
	    "dtUF".flagUF2.CEB2 OR
	    "dtUF".flagUF2.CEB2_A
	    );
	    
	    #workUF[#UF1] := "dtUF".flagUF1.Filtration AND #readyUF[#UF1];
	    #workUF[#UF2] := "dtUF".flagUF2.Filtration AND #readyUF[#UF2];
	END_REGION
	REGION Select work UF
	    "DevInWork"(ReqNumbWorkDev := #reqNumbWorkUF,
	                ReadyDev:=#readyUF,
	                WorkDev := #workUF,
	                DevCm => #cmUF,
	                ErrNotSameBound => #tErr);
	    
	    IF #cmUF[#UF1] AND "dtUF".flagUF1.StandBy THEN
	        #HandlerUF1.cmUF := "UF_CM_START";
	    END_IF;
	    IF NOT (#cmUF[#UF1]) AND "dtUF".flagUF1.Filtration THEN
	        #HandlerUF1.cmUF := "UF_CM_STOP";
	    END_IF;
	    
	    IF #cmUF[#UF2] AND "dtUF".flagUF2.StandBy THEN
	        #HandlerUF2.cmUF := "UF_CM_START";
	    END_IF;
	    IF NOT (#cmUF[#UF2]) AND "dtUF".flagUF2.Filtration THEN
	        #HandlerUF2.cmUF := "UF_CM_STOP";
	    END_IF;
	END_REGION
	REGION Block wash
	    //UF1
	    "dtUF".bUF2.HW :=
	    "dtUF".bUF2.CEB1 :=
	    "dtUF".bUF2.CEB2 :=
	    "dtUF".flagUF2.HW
	    OR "dtUF".flagUF2.HW_A
	    OR "dtUF".flagUF2.CEB1
	    OR "dtUF".flagUF2.CEB1_A
	    OR "dtUF".flagUF2.CEB2
	    OR "dtUF".flagUF2.CEB2_A;
	    
	    "dtUF".bUF2.HW_A :=
	    "dtUF".bUF2.CEB1_A :=
	    "dtUF".bUF2.CEB2_A :=
	    "dtUF".flagUF2.HW
	//    OR ("dtAnalogData".et_data["iwLT601"].Par <= "dtParmUF".minFiltrLevForWash)
	    OR "dtUF".flagUF2.HW_A
	    OR "dtUF".flagUF2.CEB1
	    OR "dtUF".flagUF2.CEB1_A
	    OR "dtUF".flagUF2.CEB2
	    OR "dtUF".flagUF2.CEB2_A;
	
	    //UF2
	    "dtUF".bUF2.HW :=
	    "dtUF".bUF2.CEB1 :=
	    "dtUF".bUF2.CEB2 :=
	    "dtUF".flagUF1.HW
	    OR "dtUF".flagUF1.HW_A
	    OR "dtUF".flagUF1.CEB1
	    OR "dtUF".flagUF1.CEB1_A
	    OR "dtUF".flagUF1.CEB2
	    OR "dtUF".flagUF1.CEB2_A;
	    
	    "dtUF".bUF2.HW_A :=
	    "dtUF".bUF2.CEB1_A :=
	    "dtUF".bUF2.CEB2_A :=
	    "dtUF".flagUF1.HW
	//   OR ("dtAnalogData".et_data["iwLT601"].Par <= "dtParmUF".minFiltrLevForWash)
	    OR "dtUF".flagUF1.HW_A
	    OR "dtUF".flagUF1.CEB1
	    OR "dtUF".flagUF1.CEB1_A
	    OR "dtUF".flagUF1.CEB2
	    OR "dtUF".flagUF1.CEB2_A;
	END_REGION
	
	REGION UF handlers
	    #HandlerUF1(// HDP := ("dtAnalogData".et_data["iwPT502"].Par - "dtAnalogData".et_data["iwPT503"].Par) >= "dtParmUF".valHDP_ForHW,
	                otherDeviceAvaible := #readyUF[#UF2],
	                otherDeviceInFiltration := "dtUF".flagUF2.Filtration,
	                filtrationTimeMin := "dtParmUF".filtrationTime,
	                flagUF := "dtUF".flagUF1,
	                delayHDP := "dtParmUF".delayHDP,
	                maxNumbHW_ByHDP := "dtParmUF".maxNumbHW_ByHDP,
	                inValve_1 => "dtAV".DVA503.cmAuto,
	                backFiltrValve_4 => "dtAV".DVA512.cmAuto,
	                upDrainValve_7 => "dtAV".DVA507.cmAuto,
	                drainTankValve_8 => "dtAV".DVA508.cmAuto,
	                drainValve_9 => "dtAV".DVA509.cmAuto,
	                airValve_10 => "dtAV".DVA501.cmAuto,
	                counters:="dtUF".countersUF1,
	                bUF:="dtUF".bUF1,
	                HW_ToCEB1 := "dtParmUF".HW_ToCEB1,
	                HW_ToCEB2 := "dtParmUF".HW_ToCEB2,
	                SoftStopSeq := "dtUfSeq".SOFT_STOP_UF1);
	    #HandlerUF2(//HDP := ("dtAnalogData".et_data["iwPT505"].Par - "dtAnalogData".et_data["iwPT506"].Par) >= "dtParmUF".valHDP_ForHW,
	                otherDeviceAvaible := #readyUF[#UF1],
	                otherDeviceInFiltration := "dtUF".flagUF1.Filtration,
	                filtrationTimeMin := "dtParmUF".filtrationTime,
	                flagUF := "dtUF".flagUF2,
	                delayHDP := "dtParmUF".delayHDP,
	                maxNumbHW_ByHDP := "dtParmUF".maxNumbHW_ByHDP,
	                inValve_1 => "dtAV".DVA510.cmAuto,
	                backFiltrValve_4 => "dtAV".DVA506.cmAuto,
	                upDrainValve_7 => "dtAV".DVA514.cmAuto,
	                drainTankValve_8 => "dtAV".DVA515.cmAuto,
	                drainValve_9 => "dtAV".DVA516.cmAuto,
	                airValve_10 => "dtAV".DVA502.cmAuto,
	                counters:="dtUF".countersUF2,
	                bUF:="dtUF".bUF2,
	                HW_ToCEB1 := "dtParmUF".HW_ToCEB1,
	                HW_ToCEB2 := "dtParmUF".HW_ToCEB2,
	                SoftStopSeq := "dtUfSeq".SOFT_STOP_UF2);
	END_REGION
	REGION Backwash valves
	    "dtAV".DVA504.cmAuto := #HandlerUF1.ownBwValve_2 OR #HandlerUF2.otherBwValve_3;
	    "dtAV".DVA511.cmAuto := #HandlerUF2.ownBwValve_2 OR #HandlerUF1.otherBwValve_3;
	END_REGION
	REGION Filtrate valves
	    //UF1
	    "dtAV".DVA505.cmAuto := #HandlerUF1.outValve_6
	    AND NOT (#HandlerUF2.clouseOtherOutValve_5 AND ("dtUF".flagUF2.HW OR "dtUF".flagUF2.CEB1 OR "dtUF".flagUF2.CEB2));
	    //UF2
	    "dtAV".DVA513.cmAuto := #HandlerUF2.outValve_6
	    AND NOT (#HandlerUF1.clouseOtherOutValve_5 AND ("dtUF".flagUF1.HW OR "dtUF".flagUF1.CEB1 OR "dtUF".flagUF1.CEB2));
	END_REGION
	REGION Display time
	    "dtUF".parUF1.Tf := TIME_TO_UDINT(IN := #HandlerUF1.filtration.PT - #HandlerUF1.filtration.ET) / 1000;
	    "dtUF".parUF2.Tf := TIME_TO_UDINT(IN := #HandlerUF2.filtration.PT - #HandlerUF2.filtration.ET) / 1000;
	    
	    "dtUF".parUF1.Ts := TIME_TO_UINT(IN := #HandlerUF1.seq.CurTime) / 1000;
	    "dtUF".parUF2.Ts := TIME_TO_UINT(IN := #HandlerUF2.seq.CurTime) / 1000;
	END_REGION
	
	
END_FUNCTION_BLOCK

FUNCTION_BLOCK "HandlerUF"
{ S7_Optimized_Access := 'TRUE' }
VERSION : 0.1
   VAR_INPUT 
      HDP : Bool;
      otherDeviceAvaible : Bool;
      otherDeviceInFiltration : Bool;
      filtrationTimeMin : UInt;
      delayHDP : UInt;
      maxNumbHW_ByHDP : UInt;
      HW_ToCEB1 : UInt;
      HW_ToCEB2 : UInt;
   END_VAR

   VAR_OUTPUT 
      inValve_1 : Bool;
      ownBwValve_2 : Bool;
      otherBwValve_3 : Bool;
      backFiltrValve_4 : Bool;
      clouseOtherOutValve_5 : Bool;
      outValve_6 : Bool;
      upDrainValve_7 : Bool;
      drainTankValve_8 : Bool;
      drainValve_9 : Bool;
      airValve_10 : Bool;
      filtrPump_11 : Bool;
      acidDPump_12 : Bool;
      clDPump_13 : Bool;
   END_VAR

   VAR_IN_OUT 
      flagUF : "UF_FLAGS";
      counters : "UF_PARAMETRS";
      bUF : "UF_COMMANDS";
   END_VAR

   VAR 
      cmUF : Int;
      needHW : Bool;
      needCEB1 : Bool;
      needCEB2 : Bool;
      CEB1_ByHDP : Bool;
      CEB2_ByHDP : Bool;
      alarmHDP : Bool;
      seq : "Sequencer";
      filtration : "TONR_200ms";
      tmrHDP : "TON_200ms";
   END_VAR

   VAR_TEMP 
      tCmUF : Int;
      tRstFiltration : Bool;
      tHoldBW : Bool;
   END_VAR


BEGIN
	REGION Action before sequence
	    CASE #cmUF OF
	        "UF_CM_STANDBY":
	            IF NOT (#flagUF.StandBy)
	            THEN
	                "RST_UF_FLAGS"(#flagUF);
	                #flagUF.StandBy := TRUE;
	                #seq.Enable := FALSE;
	                #seq.RstStep := TRUE;
	            END_IF;
	        "UF_CM_START":
	            #seq.Seq := "dtUfSeq".START;
	            IF NOT (#flagUF.Start)
	            THEN
	                "RST_UF_FLAGS"(#flagUF);
	                #flagUF.Start := TRUE;
	                #seq.Enable := TRUE;
	                #seq.RstStep := TRUE;
	            END_IF;
	        "UF_CM_FILTRATION": //Stop sequencer in filtration (realize outside custom filtration timer)
	            IF NOT (#flagUF.Filtration)
	            THEN
	                "RST_UF_FLAGS"(#flagUF);
	                #flagUF.Filtration := TRUE;
	                #seq.Enable := FALSE;
	                #seq.Done := FALSE;
	            END_IF;
	        "UF_CM_STOP":
	            #seq.Seq := "dtUfSeq".STOP;
	            IF NOT (#flagUF.Stop)
	            THEN
	                "RST_UF_FLAGS"(#flagUF);
	                #flagUF.Stop := TRUE;
	                #seq.Enable := TRUE;
	                #seq.RstStep := TRUE;
	            END_IF;
	        "UF_CM_HW":
	            #seq.Seq := "dtUfSeq".HW;
	            IF NOT (#flagUF.HW) THEN
	                IF NOT(#bUF.HW) THEN
	                    "RST_UF_FLAGS"(#flagUF);
	                    #flagUF.HW := TRUE;
	                    #seq.Enable := TRUE;
	                    #seq.RstStep := TRUE;
	                    #tRstFiltration := TRUE;
	                END_IF;
	            END_IF;
	        "UF_CM_HW_A":
	            #seq.Seq := "dtUfSeq".HW_A;
	            IF NOT (#flagUF.HW_A) THEN
	                IF NOT(#bUF.HW) THEN
	                    "RST_UF_FLAGS"(#flagUF);
	                    #flagUF.HW_A := TRUE;
	                    #seq.Enable := TRUE;
	                    #seq.RstStep := TRUE;
	                    #tRstFiltration := TRUE;
	                END_IF;
	            END_IF;
	        "UF_CM_CEB1":
	            #seq.Seq := "dtUfSeq".CEB1;
	            IF NOT (#flagUF.CEB1) THEN
	                IF NOT(#flagUF.CEB1) THEN
	                    "RST_UF_FLAGS"(#flagUF);
	                    #flagUF.CEB1 := TRUE;
	                    #seq.Enable := TRUE;
	                    #seq.RstStep := TRUE;
	                    #tRstFiltration := TRUE;
	                END_IF;
	            END_IF;
	        "UF_CM_CEB1_A":
	            #seq.Seq := "dtUfSeq".CEB1_A;
	            IF NOT (#flagUF.CEB1_A) THEN
	                IF NOT(#flagUF.CEB1_A) THEN
	                    "RST_UF_FLAGS"(#flagUF);
	                    #flagUF.CEB1_A := TRUE;
	                    #seq.Enable := TRUE;
	                    #seq.RstStep := TRUE;
	                    #tRstFiltration := TRUE;
	                END_IF;
	            END_IF;
	        "UF_CM_CEB2":
	            #seq.Seq := "dtUfSeq".CEB2;
	            IF NOT (#flagUF.CEB2) THEN
	                IF NOT (#flagUF.CEB1) THEN
	                    "RST_UF_FLAGS"(#flagUF);
	                    #flagUF.CEB2 := TRUE;
	                    #seq.Enable := TRUE;
	                    #seq.RstStep := TRUE;
	                    #tRstFiltration := TRUE;
	                END_IF;
	            END_IF;
	        "UF_CM_CEB2_A":
	            #seq.Seq := "dtUfSeq".CEB2_A;
	            IF NOT (#flagUF.CEB2_A) THEN
	                IF NOT (#flagUF.CEB2_A) THEN
	                    "RST_UF_FLAGS"(#flagUF);
	                    #flagUF.CEB2_A := TRUE;
	                    #seq.Enable := TRUE;
	                    #seq.RstStep := TRUE;
	                    #tRstFiltration := TRUE;
	                END_IF;
	
	            END_IF;
	    END_CASE;
	END_REGION
	REGION High preassure difference
	    #tmrHDP(In := #flagUF.Filtration AND #HDP,
	            PT := "intToTime_1"(intTime := #delayHDP, select := 0));
	END_REGION
	REGION Filtration
	    #filtration(In := #flagUF.Filtration,
	                PT := "intToTime_1"(intTime := #filtrationTimeMin, select := 0),
	                R := #tRstFiltration);
	END_REGION
	REGION Hold sequencer
	    #tHoldBW := #ownBwValve_2 AND #flagUF.HW AND NOT(#otherDeviceInFiltration);
	    #seq.Hold := #tHoldBW;
	END_REGION
	REGION Sequencer
	    #seq(Dev1 => #inValve_1,
	         Dev2 => #ownBwValve_2,
	         Dev3 => #otherBwValve_3,
	         Dev4 => #backFiltrValve_4,
	         Dev5 => #clouseOtherOutValve_5,
	         Dev6 => #outValve_6,
	         Dev7 => #upDrainValve_7,
	         Dev8 => #drainTankValve_8,
	         Dev9 => #drainValve_9,
	         Dev10 => #airValve_10,
	         Dev11 => #filtrPump_11,
	         Dev12 => #acidDPump_12,
	         Dev13 => #clDPump_13);
	END_REGION
	REGION Action after sequence done
	    IF #seq.Done OR #filtration.Q OR #tmrHDP.Q THEN
	      #tCmUF := #cmUF;
	      CASE #cmUF OF
	          "UF_CM_STANDBY": // After standby -> nothing
	              ;
	          "UF_CM_START": //After start -> filtration
	              #tCmUF := "UF_CM_FILTRATION";
	          "UF_CM_FILTRATION": //After filtration...
	              IF #otherDeviceAvaible THEN //Permition for stop
	                  IF NOT (#bUF.HW OR #bUF.CEB1 OR #bUF.CEB2) THEN //Simple HW
	                      #tCmUF := "UF_CM_STOP";
	                  END_IF;
	              ELSE
	                  IF NOT (#bUF.HW_A OR #bUF.CEB1_A OR #bUF.CEB2_A) THEN // Custom HW
	                      #tCmUF := "UF_CM_STOP";
	                  END_IF;
	              END_IF;
	              IF #tCmUF = "UF_CM_STOP" THEN // only after permition
	                  IF #filtration.Q THEN //Filtration done...
	                      #counters.HDPW := 0; //RST HDP counters and flags
	                      #CEB1_ByHDP := #CEB2_ByHDP := FALSE;
	                      IF #counters.HW >= #HW_ToCEB2 THEN // -> CEB2
	                          #needCEB2 := TRUE;
	                      ELSIF #counters.HW = (#HW_ToCEB1 * (#counters.CEB1 + 1)) THEN // -> CEB1
	                          #needCEB1 := TRUE;
	                      ELSE // -> HW
	                          #needHW := TRUE;
	                      END_IF;
	                  END_IF;
	                  IF #tmrHDP.Q THEN //When high delta preassure -> HW -> max count of HW -> CEB1 -> CEB2 -> alarm
	                    #counters.HDPW += 1;
	                    IF #counters.HDPW <= #maxNumbHW_ByHDP THEN
	                        #needHW := TRUE;
	                    ELSE
	                        IF #CEB1_ByHDP THEN //Do CEB1 when counter more then max number
	                              IF #CEB2_ByHDP THEN //Do CEB2 after CEB1; Again CEB2 by HDP -> alarm
	                                #alarmHDP := TRUE;
	                            ELSE
	                                #CEB2_ByHDP := TRUE;
	                                #needCEB2 := TRUE;
	                            END_IF;
	                        ELSE
	                            #CEB1_ByHDP := TRUE;
	                            #needCEB1 := TRUE;
	                        END_IF;
	                    END_IF;
	                END_IF;
	            END_IF;
	          "UF_CM_STOP": //Stop...
	            IF #alarmHDP THEN //by HDP alarm -> standby
	                #tCmUF := "UF_CM_STANDBY";
	                #alarmHDP :=
	//                #needHW :=
	//                #needCEB1 :=
	//                #needCEB2 :=
	                #CEB1_ByHDP := 
	                #CEB2_ByHDP := FALSE;
	                #counters.HDPW := 0;
	                #flagUF.ErrHDP := TRUE;
	            ELSIF #needHW THEN //by request HW -> HW/HW_A
	                #counters.HW += 1;
	                IF #otherDeviceAvaible THEN
	                    #tCmUF := "UF_CM_HW";
	                ELSE
	                    #tCmUF := "UF_CM_HW_A";
	                END_IF;
	            ELSIF #needCEB1 THEN //by request CEB1 -> CEB1/CEB1_A
	                #counters.CEB1 += 1;
	                IF #otherDeviceAvaible THEN
	                    #tCmUF := "UF_CM_CEB1";
	                ELSE
	                    #tCmUF := "UF_CM_CEB1_A";
	                END_IF;
	            ELSIF #needCEB2 THEN //by request CEB2 -> CEB2/CEB2_A
	                #counters.HW := #counters.CEB1 := 0;
	                #counters.CEB2 += 1;
	                IF #otherDeviceAvaible THEN
	                    #tCmUF := "UF_CM_CEB2";
	                ELSE
	                    #tCmUF := "UF_CM_CEB2_A";
	                END_IF;
	            ELSE //simple stop -> standby
	                #tCmUF := "UF_CM_STANDBY";
	            END_IF;
	          "UF_CM_HW",
	          "UF_CM_HW_A": //HW -> Standby
	              #needHW := FALSE;
	              #tCmUF := "UF_CM_STANDBY";
	          "UF_CM_CEB1",
	          "UF_CM_CEB1_A": //CEB1 -> Standby
	              #needCEB1 := FALSE;
	              #tCmUF := "UF_CM_STANDBY";
	          "UF_CM_CEB2",
	          "UF_CM_CEB2_A": //CEB2 -> Standby
	              #needCEB2 := FALSE;
	              #tCmUF := "UF_CM_STANDBY";
	      END_CASE;
	      #cmUF := #tCmUF;
	    END_IF;
	END_REGION
	REGION Error flag
	    #flagUF.Err :=
	    #flagUF.ErrWork
	    OR #flagUF.ErrHW
	    OR #flagUF.ErrCEB1
	    OR #flagUF.ErrCEB2
	    OR #flagUF.ErrHDP;
	END_REGION
	
	  
END_FUNCTION_BLOCK

FUNCTION_BLOCK "Sequencer"
{ S7_Optimized_Access := 'FALSE' }
VERSION : 0.1
   VAR_OUTPUT 
      Dev1 : Bool;
      Dev2 : Bool;
      Dev3 : Bool;
      Dev4 : Bool;
      Dev5 : Bool;
      Dev6 : Bool;
      Dev7 : Bool;
      Dev8 : Bool;
      Dev9 : Bool;
      Dev10 : Bool;
      Dev11 : Bool;
      Dev12 : Bool;
      Dev13 : Bool;
      Dev14 : Bool;
      Dev15 : Bool;
      Dev16 : Bool;
      CurTime : Time;
   END_VAR

   VAR 
      Enable : Bool;
      Hold : Bool;
      Seq : "Sequence" := ([TRUE], [3(1)]);
      RstStep { S7_SetPoint := 'True'} : Bool := TRUE;
      Step : Int := "MIN_STEP_NUMB";
      Timer_IN { ExternalAccessible := 'False'; ExternalVisible := 'False'; ExternalWritable := 'False'} : Bool;
      Done : Bool;
      tmr : "TON_200ms";
   END_VAR

   VAR_TEMP 
      tAddStep : Bool;
   END_VAR


BEGIN
	// Управление 16-ю механизмами в зависимости 
	// от заданной последовательности Seq 
	
	IF #RstStep THEN
	    #Step := "MIN_STEP_NUMB";
	    #Timer_IN := FALSE;
	    #Done := FALSE;
	    #RstStep := FALSE;
	END_IF;
	
	#tmr(In := #Timer_IN,
	     PT := "intToTime_1"(intTime := #Seq.delay[#Step], select := 0));
	
	#Timer_IN := #Enable AND (NOT (#tmr.Q OR #Hold OR #Done));
	#CurTime := #tmr.PT - #tmr.ET;
	
	//Переход к след. шагу
	IF #tmr.Q AND (NOT #Hold) AND (NOT #Done) THEN
	    #Step += 1;
	END_IF;
	
	IF #Enable THEN //Пропуск шагов с нулевой задержкой
	    WHILE #Seq.delay[#Step] = 0 DO
	        IF #Step >= "MAX_STEP_NUMB" THEN
	            EXIT;
	        END_IF;
	       #Step += 1;
	    END_WHILE;
	END_IF;
	
	
	//Конец последовательности
	IF #Step >= "MAX_STEP_NUMB" THEN
	    #Done := #Enable;
	    RETURN;
	END_IF;
	
	#Dev1 := #Seq.devOn[#Step, 1];
	#Dev2 := #Seq.devOn[#Step, 2];
	#Dev3 := #Seq.devOn[#Step, 3];
	#Dev4 := #Seq.devOn[#Step, 4];
	#Dev5 := #Seq.devOn[#Step, 5];
	#Dev6 := #Seq.devOn[#Step, 6];
	#Dev7 := #Seq.devOn[#Step, 7];
	#Dev8 := #Seq.devOn[#Step, 8];
	#Dev9 := #Seq.devOn[#Step, 9];
	#Dev10 := #Seq.devOn[#Step, 10];
	#Dev11 := #Seq.devOn[#Step, 11];
	#Dev12 := #Seq.devOn[#Step, 12];
	#Dev13 := #Seq.devOn[#Step, 13];
	#Dev14 := #Seq.devOn[#Step, 14];
	#Dev15 := #Seq.devOn[#Step, 15];
	#Dev16 := #Seq.devOn[#Step, 16];
	
	
	
END_FUNCTION_BLOCK

FUNCTION "intToTime_1" : Time
{ S7_Optimized_Access := 'TRUE' }
VERSION : 0.1
   VAR_INPUT 
      intTime : Int;
      select : Int;   // 0-sec, 1-min,2-hour
   END_VAR


BEGIN
	CASE #select OF
	    0:
	        #intToTime_1 := DINT_TO_TIME(INT_TO_DINT(#intTime) * 1000);
	    1:
	        #intToTime_1 := DINT_TO_TIME(INT_TO_DINT(#intTime)* 60000);
	    2:
	        #intToTime_1 := DINT_TO_TIME(INT_TO_DINT(#intTime) * 3600000);
	    ELSE  // Statement section ELSE
	        #intToTime_1 := t#0s;
	END_CASE;
END_FUNCTION

FUNCTION_BLOCK "TONR_200ms"   // FB10, FBD
{ S7_Optimized_Access := 'TRUE' }
VERSION : 0.1
// stored: AutoNumber true, IsIECCheckEnabled false, IsRetainMemResEnabled false, MemoryReserve 100, SetENOAutomatically false, UDAEnableTagReadback false
   VAR_INPUT
      In : Bool;
      PT : Time;
      R : Bool;
   END_VAR
   VAR_OUTPUT
      ET : Time;
      Q : Bool;
   END_VAR
BEGIN

REGION Network 1: Увеличение текущего времени
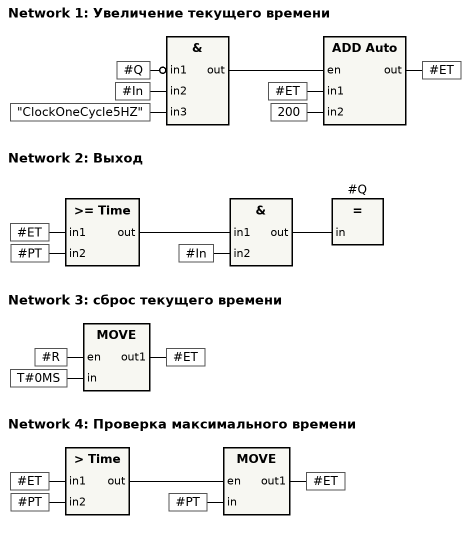
   IF NOT #Q AND #In AND "ClockOneCycle5HZ" THEN #ET := #ET + 200; END_IF;
END_REGION

REGION Network 2: Выход
   #Q := (#ET >= #PT) AND #In;
END_REGION

REGION Network 3: сброс текущего времени
   IF #R THEN #ET := T#0MS; END_IF;
END_REGION

REGION Network 4: Проверка максимального времени
   IF #ET > #PT THEN #ET := #PT; END_IF;
END_REGION
END_FUNCTION_BLOCK

FUNCTION "RST_UF_FLAGS" : Void
{ S7_Optimized_Access := 'TRUE' }
VERSION : 0.1
   VAR_IN_OUT 
      data : "UF_FLAGS";
   END_VAR


BEGIN
	#data.StandBy :=
	#data.Start :=
	#data.Stop :=
	#data.Filtration :=
	#data.HW :=
	#data.HW_A :=
	#data.CEB1 :=
	#data.CEB1_A :=
	#data.CEB2 :=
	#data.CEB2_A := FALSE;
	
END_FUNCTION

FUNCTION "DevInWork" : Void
{ S7_Optimized_Access := 'TRUE' }
VERSION : 0.1
   VAR_INPUT 
      ReqNumbWorkDev : DInt;
      ReadyDev : Array[*] of Bool;
      WorkDev : Array[*] of Bool;
   END_VAR

   VAR_OUTPUT 
      DevCm : Array[*] of Bool;
      ErrNotSameBound : Bool;
   END_VAR

   VAR_TEMP 
      tLBound : DInt;
      tUBound : DInt;
      tReqNumbWorkDev : DInt;
      i : DInt;
      tReadyDev : DInt;
      tWorkDev : DInt;
      tElemetsInArray : DInt;
   END_VAR


BEGIN
	REGION Check bounds of arrays
	    #tLBound := LOWER_BOUND(ARR := #ReadyDev, DIM := 1);
	    IF #tLBound <> LOWER_BOUND(ARR := #WorkDev, DIM := 1)
	        AND
	        #tLBound <> LOWER_BOUND(ARR := #DevCm, DIM := 1) THEN
	        #ErrNotSameBound := TRUE;
	    END_IF;
	    #tUBound := UPPER_BOUND(ARR := #ReadyDev, DIM := 1);
	    IF #tUBound <> UPPER_BOUND(ARR := #WorkDev, DIM := 1)
	        AND
	        #tUBound <> UPPER_BOUND(ARR := #DevCm, DIM := 1) THEN
	        #ErrNotSameBound := TRUE;
	    END_IF;
	    //Get count of elemets
	    FOR #i := #tLBound TO #tUBound DO
	        #tElemetsInArray += 1;
	    END_FOR;
	    
	END_REGION
	REGION Check #ReqNumbWorkDev
	    #tReqNumbWorkDev := #ReqNumbWorkDev;
	    IF #tReqNumbWorkDev < 0 THEN
	        #tReqNumbWorkDev := 0;
	    END_IF;
	    IF #tReqNumbWorkDev > #tElemetsInArray THEN
	        #tReqNumbWorkDev := #tElemetsInArray;
	    END_IF;
	END_REGION
	REGION Count ready device
	    FOR #i := #tLBound TO #tUBound DO
	        IF #ReadyDev[#i] THEN
	            #tReadyDev += 1;
	        END_IF;
	    END_FOR;
	END_REGION
	REGION Count work device
	    FOR #i := #tLBound TO #tUBound DO
	        IF #WorkDev[#i] THEN
	            #tWorkDev += 1;
	        END_IF;
	    END_FOR;
	END_REGION
	REGION Set device command
	    IF #tReqNumbWorkDev <> #tWorkDev THEN
	        FOR #i := #tLBound TO #tUBound DO
	            IF #ReadyDev[#i] THEN
	                IF #tReqNumbWorkDev > 0 THEN
	                    #DevCm[#i] := TRUE;
	                    #tReqNumbWorkDev -= 1;
	                ELSE
	                    #DevCm[#i] := FALSE;
	                END_IF;
	            ELSE
	                #DevCm[#i] := FALSE;
	            END_IF;
	        END_FOR;
	    END_IF;
	    //If bounds not same
	    IF #ErrNotSameBound THEN
	        FOR #i := #tLBound TO #tUBound DO
	            #DevCm[#i] := FALSE;
	        END_FOR;
	    END_IF;
	
	END_REGION
	
	
	
	
END_FUNCTION

ORGANIZATION_BLOCK "Cyclic interrupt"   // OB30, LAD, CyclicInterrupt
{ S7_Optimized_Access := 'TRUE' }
VERSION : 0.1
// stored: AutoNumber true, IsIECCheckEnabled false, SetENOAutomatically false
   VAR_INPUT
      Initial_Call : Bool;   // Initial call of this OB
      Event_Count : Int;   // Events discarded
   END_VAR
BEGIN

REGION Network 1: Plc analogs
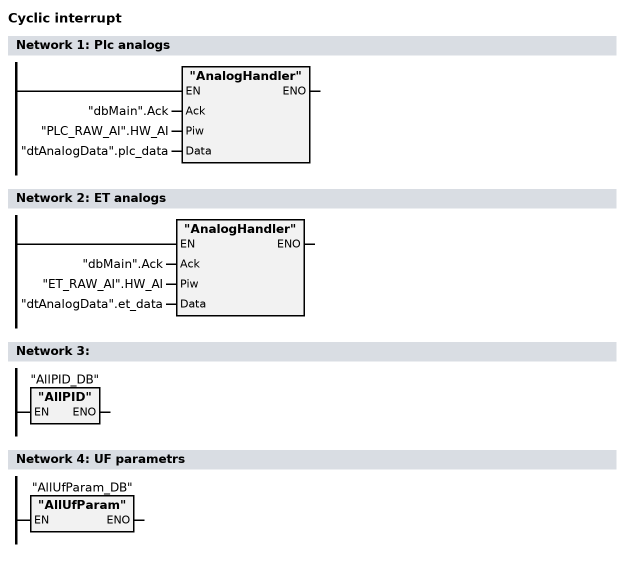
   RUNG wire#powerrail
      "AnalogHandler"(Ack := "dbMain".Ack, Piw := "PLC_RAW_AI".HW_AI, Data := "dtAnalogData".plc_data)
   END_RUNG
   // the same network as SCL:
   "AnalogHandler"(Ack := "dbMain".Ack, Piw := "PLC_RAW_AI".HW_AI, Data := "dtAnalogData".plc_data);
END_REGION

REGION Network 2: ET analogs
   RUNG wire#powerrail
      "AnalogHandler"(Ack := "dbMain".Ack, Piw := "ET_RAW_AI".HW_AI, Data := "dtAnalogData".et_data)
   END_RUNG
   // the same network as SCL:
   "AnalogHandler"(Ack := "dbMain".Ack, Piw := "ET_RAW_AI".HW_AI, Data := "dtAnalogData".et_data);
END_REGION

REGION Network 3
   RUNG wire#powerrail
      "AllPID_DB"()
   END_RUNG
   // the same network as SCL:
   "AllPID_DB"();   // "AllPID"
END_REGION

REGION Network 4: UF parametrs
   RUNG wire#powerrail
      "AllUfParam_DB"()
   END_RUNG
   // the same network as SCL:
   "AllUfParam_DB"();   // "AllUfParam"
END_REGION
END_ORGANIZATION_BLOCK

FUNCTION "AnalogHandler" : Void   // FC1, FBD
{ S7_Optimized_Access := 'TRUE' }
VERSION : 0.1
// stored: AutoNumber true, IsIECCheckEnabled false, SetENOAutomatically false, UDAEnableTagReadback false
   VAR_INPUT
      Ack : Bool;
      Piw : Array[*] of Int;
   END_VAR
   VAR_IN_OUT
      Data : Array[*] of "Ai";
   END_VAR
   VAR_TEMP
      tLb : Int;
      tUb : Int;
      i : Int;
   END_VAR
   VAR CONSTANT
      ERROR : Word := 16#01;
      BAD_PARAMETRS : Word := 16#02;
      HARDWARE_FAULT : Word := 16#04;
      SIMULATION : Word := 16#08;
      EMERGENCY_MIN : Word := 16#10;
      WARNING_MIN : Word := 16#20;
      WARNING_MAX : Word := 16#40;
      EMERGENCY_MAX : Word := 16#80;
   END_VAR
BEGIN

REGION Network 1 (SCL)
   #tLb := DINT_TO_INT(LOWER_BOUND(ARR := #Data, DIM := 1));
   #tUb := DINT_TO_INT(UPPER_BOUND(ARR := #Data, DIM := 1));

   FOR #i := #tLb TO #tUb DO
       #Data[#i].Par_code := #Piw[#i];
       #Data[#i].Par_mA := 4.0 + 16.0 * INT_TO_REAL(#Data[#i].Par_code) / 27648.0;

       IF #Data[#i].SimEnable THEN
           #Data[#i].badParam := #Data[#i].wireBreak := #Data[#i].overFlow := FALSE;
       ELSE
           #Data[#i].badParam := #Data[#i].rngUpLm < #Data[#i].rngLwLm;
           #Data[#i].wireBreak := #Data[#i].Par_code < -4866;//1.185 mA
           #Data[#i].overFlow := #Data[#i].Par_code > 32511; //22.81 mA
       END_IF;
       #Data[#i].Err :=
       #Data[#i].badParam OR
       #Data[#i].wireBreak OR
       #Data[#i].overFlow;

       IF #Data[#i].SimEnable THEN
           #Data[#i].Par := #Data[#i].SimValue;
       ELSE
           IF NOT #Data[#i].Err THEN
               #Data[#i].Par := #Data[#i].rngLwLm + INT_TO_REAL(#Data[#i].Par_code) * (#Data[#i].rngUpLm - #Data[#i].rngLwLm) / 27648.0;
               IF #Data[#i].disableParLessZero AND #Data[#i].Par < 0.0 THEN
                   #Data[#i].Par := 0.0;
               END_IF;
           ELSE
               #Data[#i].Par := 0;
           END_IF;
       END_IF;
       //Flags
       IF #Data[#i].Err THEN
           "setFlags"(enCondition := FALSE,
                      condition := #Data[#i].Par < #Data[#i].emrMin,
                      setTimerVal := #Data[#i].emrMinTime,
                      curFlag := #Data[#i].curEmMin,
                      mainFlag := #Data[#i].emMin,
                      timerVal := #Data[#i].curTimeEmrMin);
           "setFlags"(enCondition := FALSE,
                      condition := #Data[#i].Par > #Data[#i].emrMax,
                      setTimerVal := #Data[#i].emrMaxTime,
                      curFlag := #Data[#i].curEmMax,
                      mainFlag := #Data[#i].emMax,
                      timerVal := #Data[#i].curTimeEmrMax);
           "setFlags"(enCondition := FALSE,
                      condition := #Data[#i].Par < #Data[#i].wrnMin,
                      setTimerVal := #Data[#i].wrnMinTime,
                      curFlag := #Data[#i].curWnMin,
                      mainFlag := #Data[#i].wnMin,
                      timerVal := #Data[#i].curTimeWrnMin);
           "setFlags"(enCondition := FALSE,
                      condition := #Data[#i].Par > #Data[#i].wrnMax,
                      setTimerVal := #Data[#i].wrnMaxTime,
                      curFlag := #Data[#i].curWnMax,
                      mainFlag := #Data[#i].wnMax,
                      timerVal := #Data[#i].curTimeWrnMax);
           ELSE
           "setFlags"(enCondition:=#Data[#i].emMin_En,
                      condition:=#Data[#i].Par < #Data[#i].emrMin,
                      setTimerVal:=#Data[#i].emrMinTime,
                      curFlag:=#Data[#i].curEmMin,
                      mainFlag:=#Data[#i].emMin,
                      timerVal:=#Data[#i].curTimeEmrMin);
           "setFlags"(enCondition := #Data[#i].emMax_En,
                      condition := #Data[#i].Par > #Data[#i].emrMax,
                      setTimerVal := #Data[#i].emrMaxTime,
                      curFlag := #Data[#i].curEmMax,
                      mainFlag := #Data[#i].emMax,
                      timerVal := #Data[#i].curTimeEmrMax);
           "setFlags"(enCondition := #Data[#i].wrnMin_En,
                      condition := #Data[#i].Par < #Data[#i].wrnMin,
                      setTimerVal := #Data[#i].wrnMinTime,
                      curFlag := #Data[#i].curWnMin,
                      mainFlag := #Data[#i].wnMin,
                      timerVal := #Data[#i].curTimeWrnMin);
           "setFlags"(enCondition := #Data[#i].wrnMax_En,
                      condition := #Data[#i].Par > #Data[#i].wrnMax,
                      setTimerVal := #Data[#i].wrnMaxTime,
                      curFlag := #Data[#i].curWnMax,
                      mainFlag := #Data[#i].wnMax,
                      timerVal := #Data[#i].curTimeWrnMax);
       END_IF;
       //Ack
   //    #Data[#i].ackAll := #Ack;
       IF #Data[#i].modeAck THEN
           IF #Data[#i].ackAll THEN
               #Data[#i].emMin := #Data[#i].emMax := #Data[#i].wnMin := #Data[#i].wnMax := FALSE;
               #Data[#i].curTimeEmrMin := #Data[#i].curTimeEmrMax := #Data[#i].curTimeWrnMin := #Data[#i].curTimeWrnMax := 0;
           END_IF;
           IF (#Data[#i].ack AND 16#10) > 0 THEN
               #Data[#i].emMin := FALSE;
               #Data[#i].curTimeEmrMin := 0;
               #Data[#i].ack := #Data[#i].ack AND NOT(DWORD_TO_BYTE(#EMERGENCY_MIN));
           END_IF;
           IF (#Data[#i].ack AND 16#80) > 0 THEN
               #Data[#i].emMax := FALSE;
               #Data[#i].curTimeEmrMax := 0;
               #Data[#i].ack := #Data[#i].ack AND NOT(DWORD_TO_BYTE(#EMERGENCY_MAX));
           END_IF;
       ELSE
           IF NOT #Data[#i].curEmMin THEN
               #Data[#i].emMin := FALSE;
           END_IF;
           IF NOT #Data[#i].curEmMax THEN
               #Data[#i].emMax := FALSE;
           END_IF;
       END_IF;
       //Rst warning flags after normalization value
       IF NOT #Data[#i].curWnMin THEN
           #Data[#i].wnMin := FALSE;
       END_IF;
       IF NOT #Data[#i].curWnMax THEN
           #Data[#i].wnMax := FALSE;
       END_IF;
       //States:
       "setState"(condition:= NOT #Data[#i].Err,
                  hexVal:=#ERROR,
                  state:=#Data[#i].State);
       "setState"(condition := #Data[#i].badParam,
                  hexVal := #BAD_PARAMETRS,
                  state := #Data[#i].State);
       "setState"(condition := #Data[#i].wireBreak OR #Data[#i].overFlow,
                  hexVal := #HARDWARE_FAULT,
                  state := #Data[#i].State);
       "setState"(condition := #Data[#i].SimEnable,
                  hexVal := #SIMULATION,
                  state := #Data[#i].State);
       "setState"(condition := #Data[#i].emMin,
                  hexVal := #EMERGENCY_MIN,
                  state := #Data[#i].State);
       "setState"(condition := #Data[#i].wnMin,
                  hexVal := #WARNING_MIN,
                  state := #Data[#i].State);
       "setState"(condition := #Data[#i].wnMax,
                  hexVal := #WARNING_MAX,
                  state := #Data[#i].State);
       "setState"(condition := #Data[#i].emMax,
                  hexVal := #EMERGENCY_MAX,
                  state := #Data[#i].State);
   END_FOR;
END_REGION
END_FUNCTION

FUNCTION_BLOCK "AllPID"   // FB3, FBD
{ S7_Optimized_Access := 'TRUE' }
VERSION : 0.1
// stored: AutoNumber true, IsIECCheckEnabled false, IsRetainMemResEnabled false, MemoryReserve 100, SetENOAutomatically false, UDAEnableTagReadback false
   VAR
      P30x { S7_SetPoint := 'True'} : "PID_Pump2Pu1Fc";
   END_VAR
BEGIN

REGION Network 1
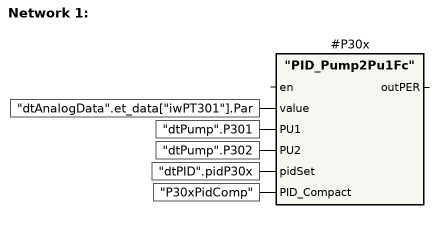
   #P30x(value := "dtAnalogData".et_data["iwPT301"].Par,   // "PID_Pump2Pu1Fc"
         PU1 := "dtPump".P301,
         PU2 := "dtPump".P302,
         pidSet := "dtPID".pidP30x,
         PID_Compact := "P30xPidComp");
END_REGION
END_FUNCTION_BLOCK

FUNCTION_BLOCK "PID_Pump2Pu1Fc"   // FB59, FBD
{ S7_Optimized_Access := 'TRUE' }
VERSION : 0.1
// stored: AutoNumber true, IsIECCheckEnabled false, IsRetainMemResEnabled false, MemoryReserve 100, SetENOAutomatically false, UDAEnableTagReadback false
   VAR_INPUT
      value : Real;
      PU1 : "Pump";
      PU2 : "Pump";
   END_VAR
   VAR_OUTPUT
      outPER : Int;
   END_VAR
   VAR_IN_OUT
      pidSet : "setPID";
      PID_Compact : PID_Compact;
   END_VAR
   VAR
      pTrigAutoMode : Bool;
      pTrigManualMode : Bool;
      pTrigCmAuto1 : Bool;
      pTrigCmAuto2 : Bool;
      nTrigCmAuto1 : Bool;
      nTrigCmAuto2 : Bool;
      pTrigFix : Bool;
      nTrigFix : Bool;
      pTrigFreez : Bool;
      nTrigFreez : Bool;
      pTrigCmHand : Bool;
      nTrigCmHand : Bool;
   END_VAR
   VAR_TEMP   // added for the SCL form of the ladder/FBD networks
      _w1 : Bool;
      _w2 : Bool;
      _w3 : Bool;
      _w4 : Bool;
      _w5 : Bool;
      _w6 : Bool;
      _w7 : Bool;
      _w8 : Bool;
      _w9 : Bool;
      _w10 : Bool;
   END_VAR
BEGIN

REGION Network 1: Интеграл
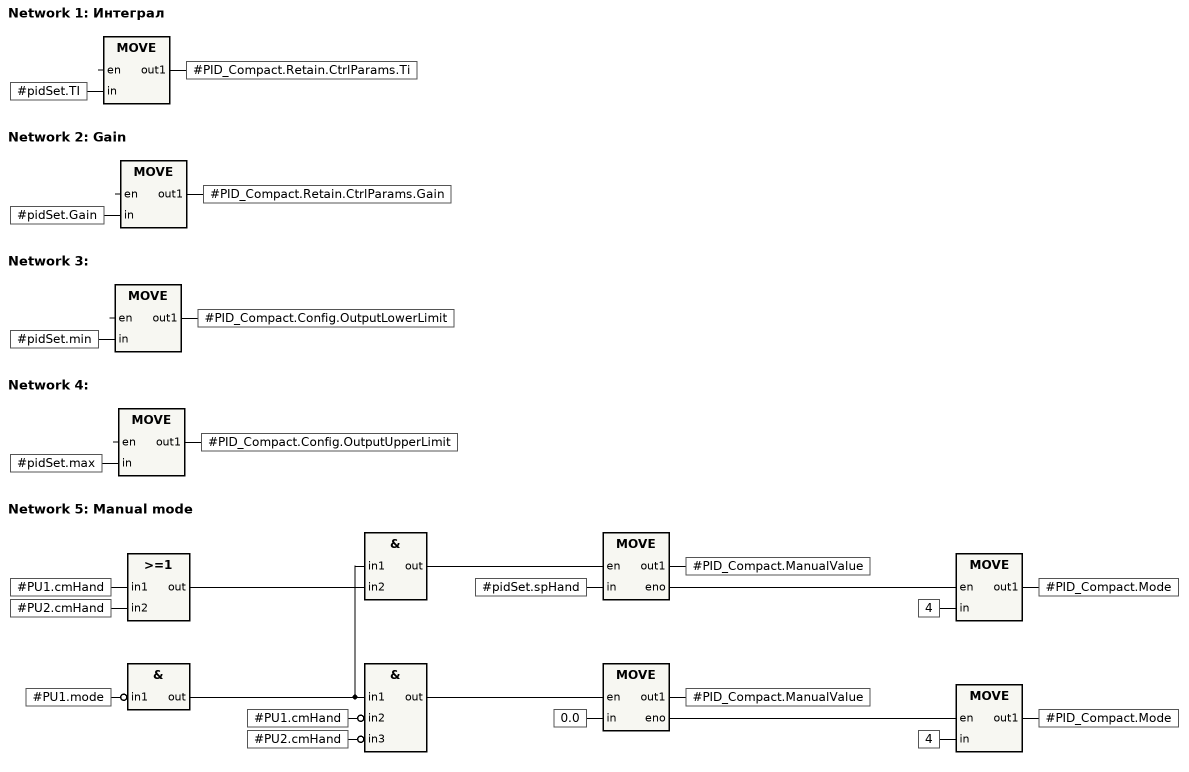
   #PID_Compact.Retain.CtrlParams.Ti := #pidSet.TI;
END_REGION

REGION Network 2: Gain
   #PID_Compact.Retain.CtrlParams.Gain := #pidSet.Gain;
END_REGION

REGION Network 3
   #PID_Compact.Config.OutputLowerLimit := #pidSet.min;
END_REGION

REGION Network 4
   #PID_Compact.Config.OutputUpperLimit := #pidSet.max;
END_REGION

REGION Network 5: Manual mode
   IF NOT #PU1.mode AND (#PU1.cmHand OR #PU2.cmHand) THEN
       #PID_Compact.ManualValue := #pidSet.spHand;
       #PID_Compact.Mode := 4;
   END_IF;
   IF NOT #PU1.mode AND NOT #PU1.cmHand AND NOT #PU2.cmHand THEN
       #PID_Compact.ManualValue := 0.0;
       #PID_Compact.Mode := 4;
   END_IF;
END_REGION

REGION Network 6: Auto mode
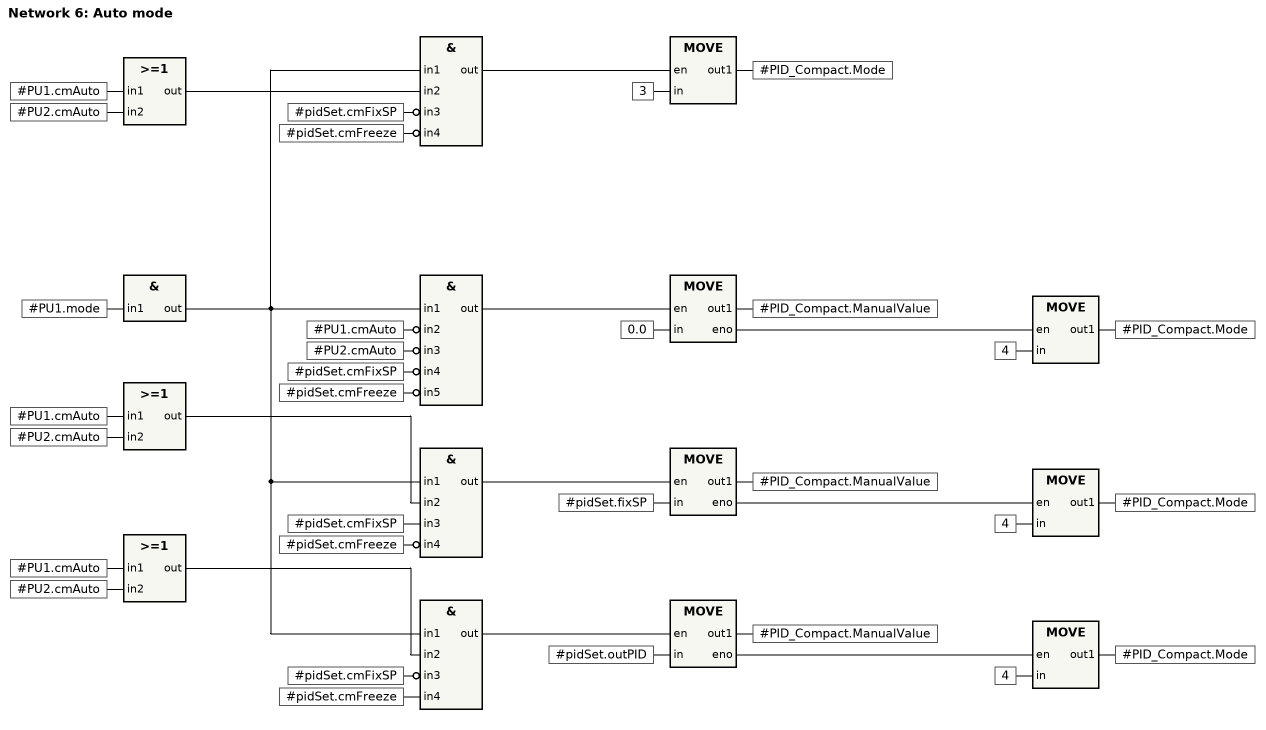
   IF #PU1.mode AND (#PU1.cmAuto OR #PU2.cmAuto) AND NOT #pidSet.cmFixSP AND NOT #pidSet.cmFreeze THEN
       #PID_Compact.Mode := 3;
   END_IF;
   IF #PU1.mode AND NOT #PU1.cmAuto AND NOT #PU2.cmAuto AND NOT #pidSet.cmFixSP AND NOT #pidSet.cmFreeze THEN
       #PID_Compact.ManualValue := 0.0;
       #PID_Compact.Mode := 4;
   END_IF;
   IF #PU1.mode AND (#PU1.cmAuto OR #PU2.cmAuto) AND #pidSet.cmFixSP AND NOT #pidSet.cmFreeze THEN
       #PID_Compact.ManualValue := #pidSet.fixSP;
       #PID_Compact.Mode := 4;
   END_IF;
   IF #PU1.mode AND (#PU1.cmAuto OR #PU2.cmAuto) AND NOT #pidSet.cmFixSP AND #pidSet.cmFreeze THEN
       #PID_Compact.ManualValue := #pidSet.outPID;
       #PID_Compact.Mode := 4;
   END_IF;
END_REGION

REGION Network 7: Set modeActivate
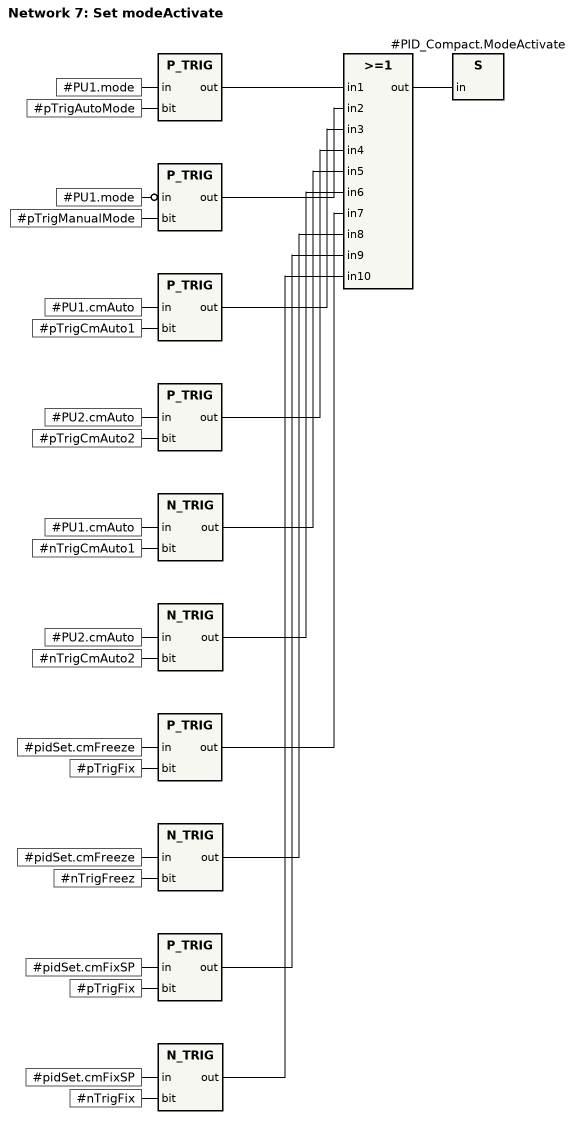
   #_w1 := #PU1.mode AND NOT #pTrigAutoMode;   // rising edge
   #pTrigAutoMode := #PU1.mode;
   #_w2 := NOT #PU1.mode AND NOT #pTrigManualMode;   // rising edge
   #pTrigManualMode := NOT #PU1.mode;
   #_w3 := #PU1.cmAuto AND NOT #pTrigCmAuto1;   // rising edge
   #pTrigCmAuto1 := #PU1.cmAuto;
   #_w4 := #PU2.cmAuto AND NOT #pTrigCmAuto2;   // rising edge
   #pTrigCmAuto2 := #PU2.cmAuto;
   #_w5 := NOT #PU1.cmAuto AND #nTrigCmAuto1;   // falling edge
   #nTrigCmAuto1 := #PU1.cmAuto;
   #_w6 := NOT #PU2.cmAuto AND #nTrigCmAuto2;   // falling edge
   #nTrigCmAuto2 := #PU2.cmAuto;
   #_w7 := #pidSet.cmFreeze AND NOT #pTrigFix;   // rising edge
   #pTrigFix := #pidSet.cmFreeze;
   #_w8 := NOT #pidSet.cmFreeze AND #nTrigFreez;   // falling edge
   #nTrigFreez := #pidSet.cmFreeze;
   #_w9 := #pidSet.cmFixSP AND NOT #pTrigFix;   // rising edge
   #pTrigFix := #pidSet.cmFixSP;
   #_w10 := NOT #pidSet.cmFixSP AND #nTrigFix;   // falling edge
   #nTrigFix := #pidSet.cmFixSP;
   IF #_w1 OR #_w2 OR #_w3 OR #_w4 OR #_w5 OR #_w6 OR #_w7 OR #_w8 OR #_w9 OR #_w10 THEN
       #PID_Compact.ModeActivate := TRUE;
   END_IF;
END_REGION

REGION Network 8
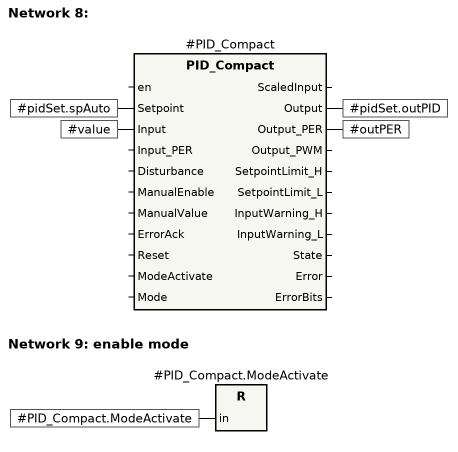
   #PID_Compact(Setpoint := #pidSet.spAuto, Input := #value, Output => #pidSet.outPID, Output_PER => #outPER);   // PID_Compact
END_REGION

REGION Network 9: enable mode
   IF #PID_Compact.ModeActivate THEN #PID_Compact.ModeActivate := FALSE; END_IF;
END_REGION
END_FUNCTION_BLOCK

FUNCTION_BLOCK "AllUfParam"
{ S7_Optimized_Access := 'TRUE' }
VERSION : 0.1
   VAR 
      mSec : USInt;
      sec : UInt;
      inVolumeUF1 : Real;
      inVolumeUF2 : Real;
      outVolumeUF1 : Real;
      outVolumeUF2 : Real;
   END_VAR

   VAR CONSTANT 
      RECOVERY_PERIOD : UInt := 7200;
   END_VAR


BEGIN
	//Cycle Time is 0.1 sec
	//
	REGION Recovery timer
	    #mSec += 1;
	    IF #mSec >= 10 THEN
	        #mSec := 0;
	        #sec += 1;
	    END_IF;
	    IF #sec >= #RECOVERY_PERIOD THEN
	        #sec := 0;
	        #inVolumeUF1 := "dbVolumeCounters".FM501.all;
	        #inVolumeUF2 := "dbVolumeCounters".FM502.all;
	        // #outVolumeUF1 := ;
	        // #outVolumeUF2 := ;
	    END_IF;
	END_REGION
	"dtUF".parUF1.flux := "Flux"("inFlow(m3/h)" := "dtAnalogData".et_data["iwFM501"].Par,
	                             "Sfiltr(m2)" := "dtUF".parUF1.Sf);
	"dtUF".parUF2.flux := "Flux"("inFlow(m3/h)" := "dtAnalogData".et_data["iwFM502"].Par,
	                             "Sfiltr(m2)" := "dtUF".parUF2.Sf);
	"dtUF".parUF1.dP := "dtAnalogData".et_data["iwPT502"].Par - "dtAnalogData".et_data["iwPT503"].Par;
	"dtUF".parUF2.dP := "dtAnalogData".et_data["iwPT505"].Par - "dtAnalogData".et_data["iwPT506"].Par;
	"dtUF".parUF1.Rec := "Recovery"(inVolume := #inVolumeUF1, outVolume := #outVolumeUF1);
	"dtUF".parUF2.Rec := "Recovery"(inVolume := #inVolumeUF2, outVolume := #outVolumeUF2);
END_FUNCTION_BLOCK

FUNCTION "Recovery" : Real
{ S7_Optimized_Access := 'TRUE' }
VERSION : 0.1
   VAR_INPUT 
      inVolume : Real;
      outVolume : Real;
   END_VAR


BEGIN
	IF (#inVolume <= 0) OR (#outVolume <= 0) THEN
	    #Recovery := 0;
	    RETURN;
	ELSE
	    #Recovery := (#outVolume / #inVolume) * 100;
	END_IF;
END_FUNCTION

FUNCTION_BLOCK "tmr200ms"   // FB9, FBD
{ S7_Optimized_Access := 'TRUE' }
VERSION : 0.1
// stored: AutoNumber true, IsIECCheckEnabled false, IsRetainMemResEnabled false, MemoryReserve 100, SetENOAutomatically false, UDAEnableTagReadback false
   VAR_INPUT
      In : Bool;
      PT : Time;
   END_VAR
   VAR_OUTPUT
      ET : Time;
      Q : Bool;
   END_VAR
BEGIN

REGION Network 1: Увеличение текущего времени
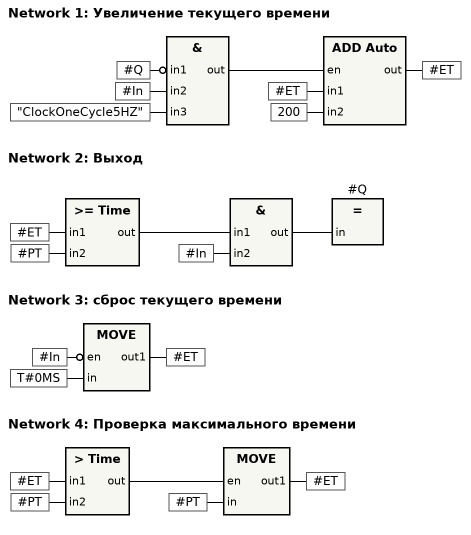
   IF NOT #Q AND #In AND "ClockOneCycle5HZ" THEN #ET := #ET + 200; END_IF;
END_REGION

REGION Network 2: Выход
   #Q := (#ET >= #PT) AND #In;
END_REGION

REGION Network 3: сброс текущего времени
   IF NOT #In THEN #ET := T#0MS; END_IF;
END_REGION

REGION Network 4: Проверка максимального времени
   IF #ET > #PT THEN #ET := #PT; END_IF;
END_REGION
END_FUNCTION_BLOCK

FUNCTION "setFlags" : Void   // FC2, FBD
{ S7_Optimized_Access := 'TRUE' }
VERSION : 0.1
// stored: AutoNumber true, IsIECCheckEnabled false, SetENOAutomatically false, UDAEnableTagReadback false
   VAR_INPUT
      enCondition : Bool;
      condition : Bool;
      setTimerVal : Real;
   END_VAR
   VAR_IN_OUT
      curFlag : Bool;
      mainFlag : Bool;
      timerVal : Real;
   END_VAR
BEGIN

REGION Network 1 (SCL)

   #curFlag := #enCondition AND #condition;

   IF NOT #curFlag THEN
       #timerVal := 0;
   END_IF;

   IF #curFlag AND #timerVal < #setTimerVal THEN
       #timerVal += 0.1;
   END_IF;

   IF #timerVal >= #setTimerVal THEN
       #mainFlag := TRUE;
   END_IF;
END_REGION
END_FUNCTION

FUNCTION "setState" : Void   // FC3, FBD
{ S7_Optimized_Access := 'TRUE' }
VERSION : 0.1
// stored: AutoNumber true, IsIECCheckEnabled false, SetENOAutomatically false, UDAEnableTagReadback false
   VAR_INPUT
      condition : Bool;
      hexVal : Word;
   END_VAR
   VAR_IN_OUT
      state : Word;
   END_VAR
BEGIN

REGION Network 1 (SCL)
   IF #condition THEN
       // Statement section IF
       #state := #state OR #hexVal;
   ELSE
       #state := #state AND NOT #hexVal;
   END_IF;
END_REGION
END_FUNCTION

FUNCTION_BLOCK "PumpAckAlarm"   // FB38, LAD
{ S7_Optimized_Access := 'TRUE' }
VERSION : 0.1
// stored: AutoNumber true, IsIECCheckEnabled false, IsRetainMemResEnabled false, MemoryReserve 100, SetENOAutomatically false, UDAEnableTagReadback false
   VAR_INPUT
      ack : Bool;
      power : Bool;
      alarmFC : Bool;
      emrStop : Bool;   // Авариный стоп 0-авария, 1-ок
      local : Bool;   // 1-местный режим
      tmrOpening_Q : Bool;
      tmrClosing_Q : Bool;
   END_VAR
   VAR_IN_OUT
      dev : "Pump";
      errService : Bool;
      ErrPower : Bool;   // Признак аварии питания
      errAlarmFc : Bool;
      ErrDis : Bool;   // Признак внешней блокировки
      errEmrStop : Bool;
      errLocal : Bool;
      errStart : Bool;
      errStop : Bool;
   END_VAR
   VAR
      InstService { S7_SetPoint := 'True'} : "DevAckSingleAlarm";
      InstPower { S7_SetPoint := 'True'} : "DevAckSingleAlarm";
      InstFc { S7_SetPoint := 'True'} : "DevAckSingleAlarm";
      InstDis { S7_SetPoint := 'True'} : "DevBlockAckSingleAlarm";
      InstEmrStop { S7_SetPoint := 'True'} : "DevAckSingleAlarm";
      InstLocal { S7_SetPoint := 'True'} : "DevAckSingleAlarm";
      InstStart { S7_SetPoint := 'True'} : "DevAckSingleAlarm";
      InstStop { S7_SetPoint := 'True'} : "DevAckSingleAlarm";
   END_VAR
BEGIN

REGION Network 1: Сервисный режим - нужно квитирование ACK
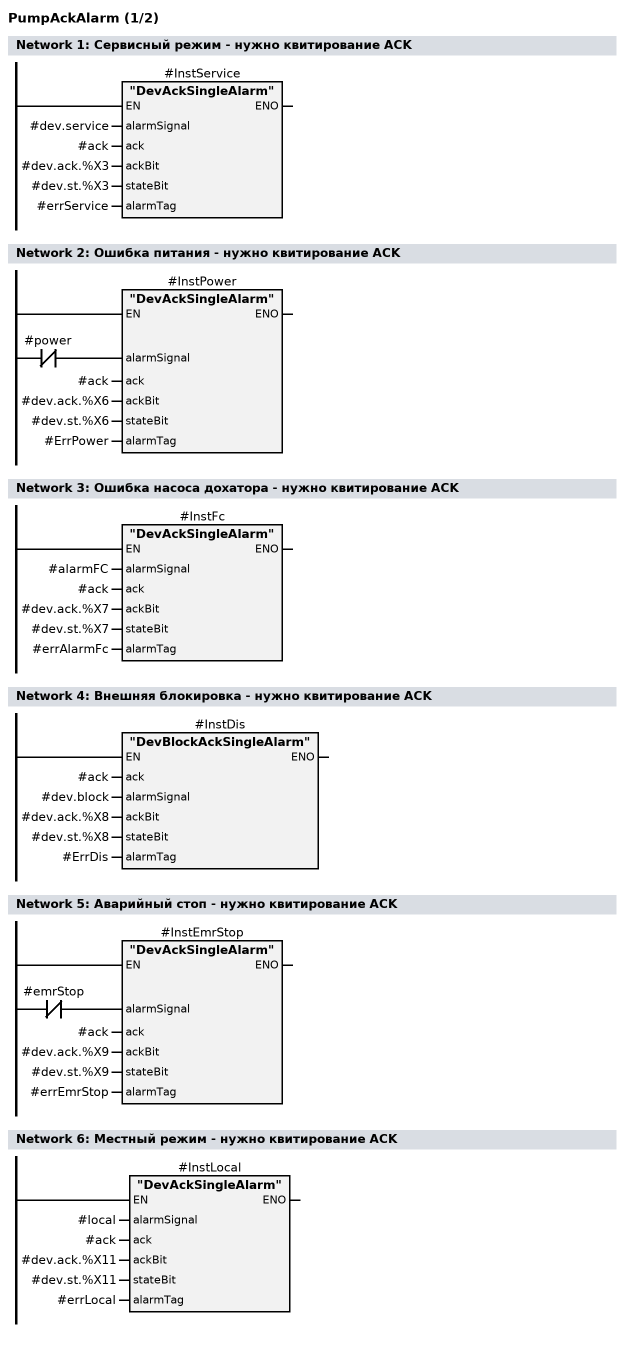
   RUNG wire#powerrail
      #InstService(alarmSignal := #dev.service, ack := #ack, ackBit := #dev.ack.%X3, stateBit := #dev.st.%X3, alarmTag := #errService)
   END_RUNG
   // the same network as SCL:
   #InstService(alarmSignal := #dev.service,   // "DevAckSingleAlarm"
                ack := #ack,
                ackBit := #dev.ack.%X3,
                stateBit := #dev.st.%X3,
                alarmTag := #errService);
END_REGION

REGION Network 2: Ошибка питания - нужно квитирование ACK
   RUNG wire#powerrail
      #InstPower(alarmSignal := wire#w1, ack := #ack, ackBit := #dev.ack.%X6, stateBit := #dev.st.%X6, alarmTag := #ErrPower)
   END_RUNG
   RUNG wire#powerrail
      I_Contact( #power )
   END_RUNG wire#w1
   // the same network as SCL:
   #InstPower(alarmSignal := NOT #power,   // "DevAckSingleAlarm"
              ack := #ack,
              ackBit := #dev.ack.%X6,
              stateBit := #dev.st.%X6,
              alarmTag := #ErrPower);
END_REGION

REGION Network 3: Ошибка насоса дохатора - нужно квитирование ACK
   RUNG wire#powerrail
      #InstFc(alarmSignal := #alarmFC, ack := #ack, ackBit := #dev.ack.%X7, stateBit := #dev.st.%X7, alarmTag := #errAlarmFc)
   END_RUNG
   // the same network as SCL:
   #InstFc(alarmSignal := #alarmFC,   // "DevAckSingleAlarm"
           ack := #ack,
           ackBit := #dev.ack.%X7,
           stateBit := #dev.st.%X7,
           alarmTag := #errAlarmFc);
END_REGION

REGION Network 4: Внешняя блокировка - нужно квитирование ACK
   RUNG wire#powerrail
      #InstDis(ack := #ack, alarmSignal := #dev.block, ackBit := #dev.ack.%X8, stateBit := #dev.st.%X8, alarmTag := #ErrDis)
   END_RUNG
   // the same network as SCL:
   #InstDis(ack := #ack,   // "DevBlockAckSingleAlarm"
            alarmSignal := #dev.block,
            ackBit := #dev.ack.%X8,
            stateBit := #dev.st.%X8,
            alarmTag := #ErrDis);
END_REGION

REGION Network 5: Аварийный стоп - нужно квитирование ACK
   RUNG wire#powerrail
      #InstEmrStop(alarmSignal := wire#w1, ack := #ack, ackBit := #dev.ack.%X9, stateBit := #dev.st.%X9, alarmTag := #errEmrStop)
   END_RUNG
   RUNG wire#powerrail
      I_Contact( #emrStop )
   END_RUNG wire#w1
   // the same network as SCL:
   #InstEmrStop(alarmSignal := NOT #emrStop,   // "DevAckSingleAlarm"
                ack := #ack,
                ackBit := #dev.ack.%X9,
                stateBit := #dev.st.%X9,
                alarmTag := #errEmrStop);
END_REGION

REGION Network 6: Местный режим - нужно квитирование ACK
   RUNG wire#powerrail
      #InstLocal(alarmSignal := #local, ack := #ack, ackBit := #dev.ack.%X11, stateBit := #dev.st.%X11, alarmTag := #errLocal)
   END_RUNG
   // the same network as SCL:
   #InstLocal(alarmSignal := #local,   // "DevAckSingleAlarm"
              ack := #ack,
              ackBit := #dev.ack.%X11,
              stateBit := #dev.st.%X11,
              alarmTag := #errLocal);
END_REGION

REGION Network 7: Состояние ошибки запуска ACK
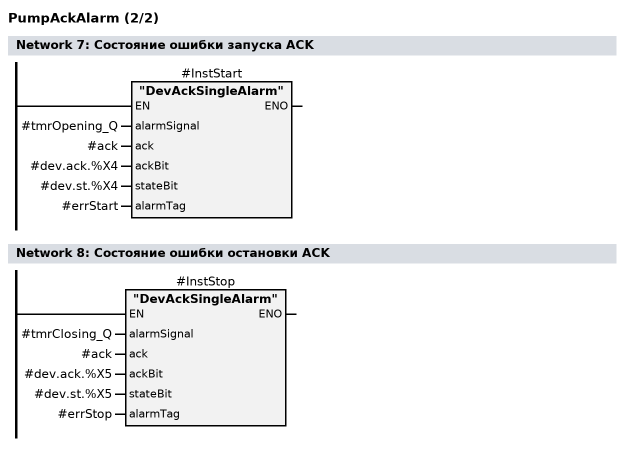
   RUNG wire#powerrail
      #InstStart(alarmSignal := #tmrOpening_Q, ack := #ack, ackBit := #dev.ack.%X4, stateBit := #dev.st.%X4, alarmTag := #errStart)
   END_RUNG
   // the same network as SCL:
   #InstStart(alarmSignal := #tmrOpening_Q,   // "DevAckSingleAlarm"
              ack := #ack,
              ackBit := #dev.ack.%X4,
              stateBit := #dev.st.%X4,
              alarmTag := #errStart);
END_REGION

REGION Network 8: Состояние ошибки остановки ACK
   RUNG wire#powerrail
      #InstStop(alarmSignal := #tmrClosing_Q, ack := #ack, ackBit := #dev.ack.%X5, stateBit := #dev.st.%X5, alarmTag := #errStop)
   END_RUNG
   // the same network as SCL:
   #InstStop(alarmSignal := #tmrClosing_Q,   // "DevAckSingleAlarm"
             ack := #ack,
             ackBit := #dev.ack.%X5,
             stateBit := #dev.st.%X5,
             alarmTag := #errStop);
END_REGION
END_FUNCTION_BLOCK

FUNCTION_BLOCK "PumpCntr"   // FB60, LAD
{ S7_Optimized_Access := 'FALSE' }
VERSION : 0.1
// #ST:
// номер бита, часло десятичное
//  0  - стоп 
// 0 1 - работа
// 1 2 - запуск
// 2 4 - остановка
// 3 8 - сервисный режим
// 4 16 - ошибка Пуска
// 5 32 - ошибка Стопа
// 6 64 - ошибка питания
// 7 128 - ошибка частотника (дозатора)
// 8 256 - Блокировка внешняя
// 9 - 512 - нажат аварийный стоп
// 10 -1024 - сборная авария
// 11 2048 - местный режим
// 12 4096
// 13 8192
// 14 16384 1-показывать кнопки ручного управления
// 15 32768 - режим 1-ручной, 0-авто (только для индкатора на скаде)
// stored: AutoNumber false, IsIECCheckEnabled false, SetENOAutomatically false, UDAEnableTagReadback false
   VAR_INPUT
      power : Bool;   // питание устройства 1-ок
      run : Bool;   // 1-работа
      emrStop : Bool;   // Авариный стоп 0-авария, 1-ок
      local : Bool;   // 1-местный режим
      alarmFC : Bool;   // 1-авария
      block1 : Bool;
      block2 : Bool;
      block3 : Bool;
      block4 : Bool;
      block5 : Bool;
      block6 : Bool;
   END_VAR
   VAR_OUTPUT
      qStart : Bool;   // пуск
   END_VAR
   VAR_IN_OUT
      dev : "Pump";
   END_VAR
   VAR DB_SPECIFIC
      ErrOC : Bool;   // Признак аварии по закрытию или открытию
      ErrPower : Bool;   // Признак аварии питания
      ErrDis : Bool;   // Признак внешней блокировки
      qON : Bool;   // Выход для управления механизмом
      tmrClosing { S7_SetPoint := 'True'} : TON_TIME;
      tmrOpening { S7_SetPoint := 'True'} : TON_TIME;
      closed : Bool;
      opened : Bool;
      closing : Bool;
      opening : Bool;
      errStart : Bool;
      errStop : Bool;
      errEmrStop : Bool;
      errAlarmFc : Bool;
      errService : Bool;
      errLocal : Bool;
      tStart : Time;
      tStop : Time;
   END_VAR
   VAR
      DpumpAckAlarm_Instance : "PumpAckAlarm";
   END_VAR
   VAR CONSTANT
      ACK_DELAY : Time := T#1s;
   END_VAR
BEGIN

REGION Network 1: Сброс состояния
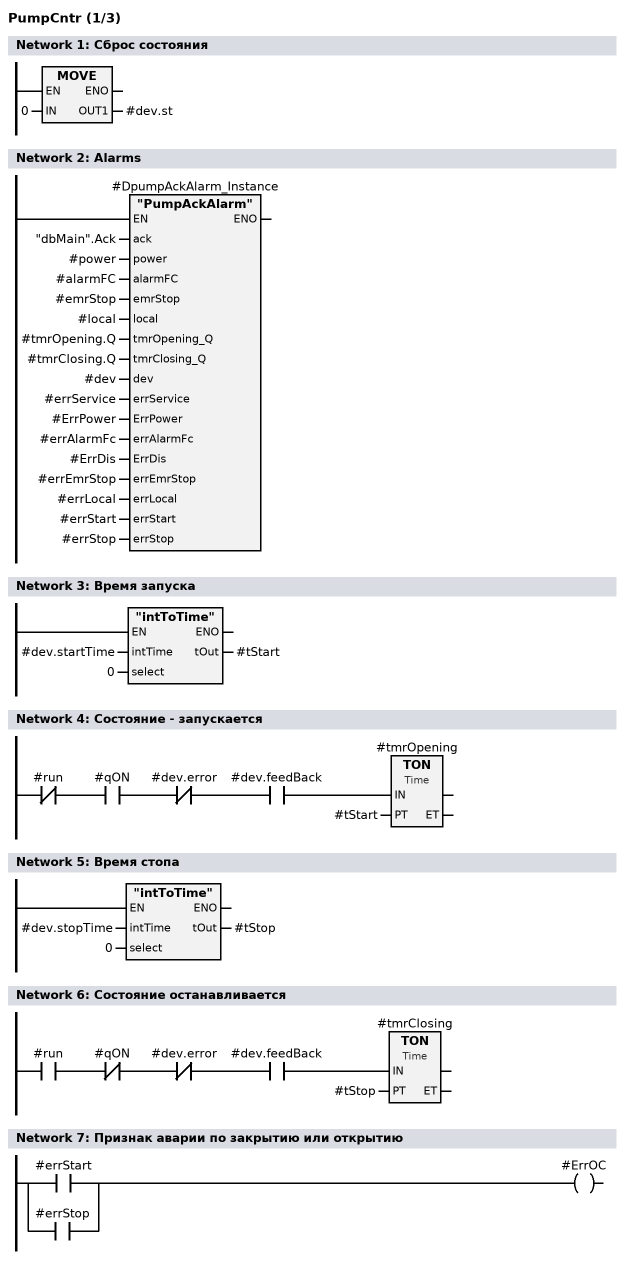
   RUNG wire#powerrail
      { S7_GenerateENO := "TRUE" } Move(in := 0, out1 => #dev.st)
   END_RUNG
   // the same network as SCL:
   #dev.st := 0;
END_REGION

REGION Network 2: Alarms
   RUNG wire#powerrail
      #DpumpAckAlarm_Instance(ack := "dbMain".Ack, power := #power, alarmFC := #alarmFC, emrStop := #emrStop, local := #local, tmrOpening_Q := #tmrOpening.Q, tmrClosing_Q := #tmrClosing.Q, dev := #dev, errService := #errService, ErrPower := #ErrPower, errAlarmFc := #errAlarmFc, ErrDis := #ErrDis, errEmrStop := #errEmrStop, errLocal := #errLocal, errStart := #errStart, errStop := #errStop)
   END_RUNG
   // the same network as SCL:
   #DpumpAckAlarm_Instance(ack := "dbMain".Ack,   // "PumpAckAlarm"
                           power := #power,
                           alarmFC := #alarmFC,
                           emrStop := #emrStop,
                           local := #local,
                           tmrOpening_Q := #tmrOpening.Q,
                           tmrClosing_Q := #tmrClosing.Q,
                           dev := #dev,
                           errService := #errService,
                           ErrPower := #ErrPower,
                           errAlarmFc := #errAlarmFc,
                           ErrDis := #ErrDis,
                           errEmrStop := #errEmrStop,
                           errLocal := #errLocal,
                           errStart := #errStart,
                           errStop := #errStop);
END_REGION

REGION Network 3: Время запуска
   RUNG wire#powerrail
      "intToTime"(intTime := #dev.startTime, select := 0, tOut => #tStart)
   END_RUNG
   // the same network as SCL:
   "intToTime"(intTime := #dev.startTime, select := 0, tOut => #tStart);
END_REGION

REGION Network 4: Состояние - запускается
   RUNG wire#powerrail
      I_Contact( #run )
      Contact( #qON )
      I_Contact( #dev.error )
      Contact( #dev.feedBack )
      { S7_Templates := "time_type := Time" } #tmrOpening.TON(pt := #tStart, et =>)
   END_RUNG
   // the same network as SCL:
   #tmrOpening(IN := NOT #run AND #qON AND NOT #dev.error AND #dev.feedBack, PT := #tStart);   // TON
END_REGION

REGION Network 5: Время стопа
   RUNG wire#powerrail
      "intToTime"(intTime := #dev.stopTime, select := 0, tOut => #tStop)
   END_RUNG
   // the same network as SCL:
   "intToTime"(intTime := #dev.stopTime, select := 0, tOut => #tStop);
END_REGION

REGION Network 6: Состояние останавливается
   RUNG wire#powerrail
      Contact( #run )
      I_Contact( #qON )
      I_Contact( #dev.error )
      Contact( #dev.feedBack )
      { S7_Templates := "time_type := Time" } #tmrClosing.TON(pt := #tStop, et =>)
   END_RUNG
   // the same network as SCL:
   #tmrClosing(IN := #run AND NOT #qON AND NOT #dev.error AND #dev.feedBack, PT := #tStop);   // TON
END_REGION

REGION Network 7: Признак аварии по закрытию или открытию
   RUNG wire#powerrail
      Contact( #errStart )
      wire#w1
      Coil( #ErrOC )
   END_RUNG
   RUNG wire#powerrail
      Contact( #errStop )
   END_RUNG wire#w1
   // the same network as SCL:
   #ErrOC := #errStart OR #errStop;
END_REGION

REGION Network 8: Сборная авария
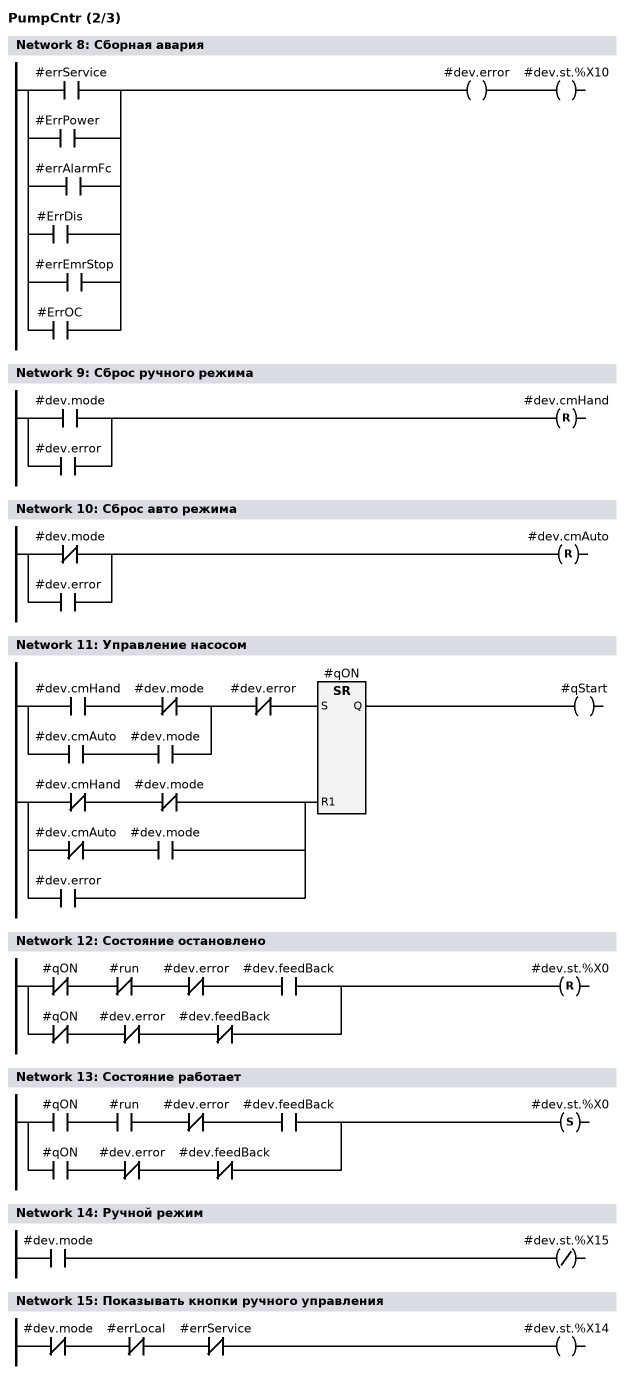
   RUNG wire#powerrail
      Contact( #errService )
      wire#w1
      Coil( #dev.error )
      Coil( #dev.st.%X10 )
   END_RUNG
   RUNG wire#powerrail
      Contact( #ErrPower )
   END_RUNG wire#w1
   RUNG wire#powerrail
      Contact( #errAlarmFc )
   END_RUNG wire#w1
   RUNG wire#powerrail
      Contact( #ErrDis )
   END_RUNG wire#w1
   RUNG wire#powerrail
      Contact( #errEmrStop )
   END_RUNG wire#w1
   RUNG wire#powerrail
      Contact( #ErrOC )
   END_RUNG wire#w1
   // the same network as SCL:
   #dev.error := #errService OR #ErrPower OR #errAlarmFc OR #ErrDis OR #errEmrStop OR #ErrOC;
   #dev.st.%X10 := #dev.error;
END_REGION

REGION Network 9: Сброс ручного режима
   RUNG wire#powerrail
      Contact( #dev.mode )
      wire#w1
      R_Coil( #dev.cmHand )
   END_RUNG
   RUNG wire#powerrail
      Contact( #dev.error )
   END_RUNG wire#w1
   // the same network as SCL:
   IF #dev.mode OR #dev.error THEN #dev.cmHand := FALSE; END_IF;
END_REGION

REGION Network 10: Сброс авто режима
   RUNG wire#powerrail
      I_Contact( #dev.mode )
      wire#w1
      R_Coil( #dev.cmAuto )
   END_RUNG
   RUNG wire#powerrail
      Contact( #dev.error )
   END_RUNG wire#w1
   // the same network as SCL:
   IF NOT #dev.mode OR #dev.error THEN #dev.cmAuto := FALSE; END_IF;
END_REGION

REGION Network 11: Управление насосом
   RUNG wire#powerrail
      Contact( #dev.cmHand )
      I_Contact( #dev.mode )
      wire#w1
      I_Contact( #dev.error )
      S_SR(operand := #qON, r1 := wire#w2)
      Coil( #qStart )
   END_RUNG
   RUNG wire#powerrail
      Contact( #dev.cmAuto )
      Contact( #dev.mode )
   END_RUNG wire#w1
   RUNG wire#powerrail
      I_Contact( #dev.cmHand )
      I_Contact( #dev.mode )
   END_RUNG wire#w2
   RUNG wire#powerrail
      I_Contact( #dev.cmAuto )
      Contact( #dev.mode )
   END_RUNG wire#w2
   RUNG wire#powerrail
      Contact( #dev.error )
   END_RUNG wire#w2
   // the same network as SCL:
   IF ((#dev.cmHand AND NOT #dev.mode) OR (#dev.cmAuto AND #dev.mode)) AND NOT #dev.error THEN
       #qON := TRUE;   // SR flip-flop
   END_IF;
   IF (NOT #dev.cmHand AND NOT #dev.mode) OR (NOT #dev.cmAuto AND #dev.mode) OR #dev.error THEN
       #qON := FALSE;
   END_IF;
   #qStart := #qON;
END_REGION

REGION Network 12: Состояние остановлено
   RUNG wire#powerrail
      I_Contact( #qON )
      I_Contact( #run )
      I_Contact( #dev.error )
      Contact( #dev.feedBack )
      wire#w1
      R_Coil( #dev.st.%X0 )
   END_RUNG
   RUNG wire#powerrail
      I_Contact( #qON )
      I_Contact( #dev.error )
      I_Contact( #dev.feedBack )
   END_RUNG wire#w1
   // the same network as SCL:
   IF (NOT #qON AND NOT #run AND NOT #dev.error AND #dev.feedBack) OR (NOT #qON AND NOT #dev.error AND NOT #dev.feedBack) THEN
       #dev.st.%X0 := FALSE;
   END_IF;
END_REGION

REGION Network 13: Состояние работает
   RUNG wire#powerrail
      Contact( #qON )
      Contact( #run )
      I_Contact( #dev.error )
      Contact( #dev.feedBack )
      wire#w1
      S_Coil( #dev.st.%X0 )
   END_RUNG
   RUNG wire#powerrail
      Contact( #qON )
      I_Contact( #dev.error )
      I_Contact( #dev.feedBack )
   END_RUNG wire#w1
   // the same network as SCL:
   IF (#qON AND #run AND NOT #dev.error AND #dev.feedBack) OR (#qON AND NOT #dev.error AND NOT #dev.feedBack) THEN
       #dev.st.%X0 := TRUE;
   END_IF;
END_REGION

REGION Network 14: Ручной режим
   RUNG wire#powerrail
      Contact( #dev.mode )
      I_Coil( #dev.st.%X15 )
   END_RUNG
   // the same network as SCL:
   #dev.st.%X15 := NOT #dev.mode;
END_REGION

REGION Network 15: Показывать кнопки ручного управления
   RUNG wire#powerrail
      I_Contact( #dev.mode )
      I_Contact( #errLocal )
      I_Contact( #errService )
      Coil( #dev.st.%X14 )
   END_RUNG
   // the same network as SCL:
   #dev.st.%X14 := NOT #dev.mode AND NOT #errLocal AND NOT #errService;
END_REGION

REGION Network 16: Программный выход запуска насоса
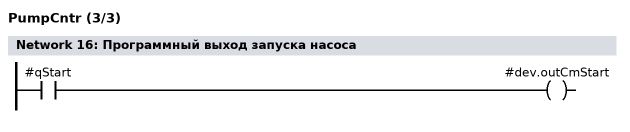
   RUNG wire#powerrail
      Contact( #qStart )
      Coil( #dev.outCmStart )
   END_RUNG
   // the same network as SCL:
   #dev.outCmStart := #qStart;
END_REGION
END_FUNCTION_BLOCK

FUNCTION_BLOCK "VolumeCounter"   // FB65, FBD
{ S7_Optimized_Access := 'TRUE' }
VERSION : 0.1
// stored: AutoNumber true, IsIECCheckEnabled false, IsRetainMemResEnabled false, MemoryReserve 100, SetENOAutomatically false, UDAEnableTagReadback false
   VAR_INPUT
      puls : Bool;
      nextHour : Bool;
      nextDay : Bool;
   END_VAR
   VAR_IN_OUT
      data : "FREQ_COUNTER";
   END_VAR
   VAR
      litrs : UInt;
      pTrig : Bool;
   END_VAR
   VAR CONSTANT
      FB_CALL_TIME : Real := 0.1;
   END_VAR
   VAR_TEMP   // added for the SCL form of the ladder/FBD networks
      _w1 : Bool;
   END_VAR
BEGIN

REGION Network 1: Add to counter
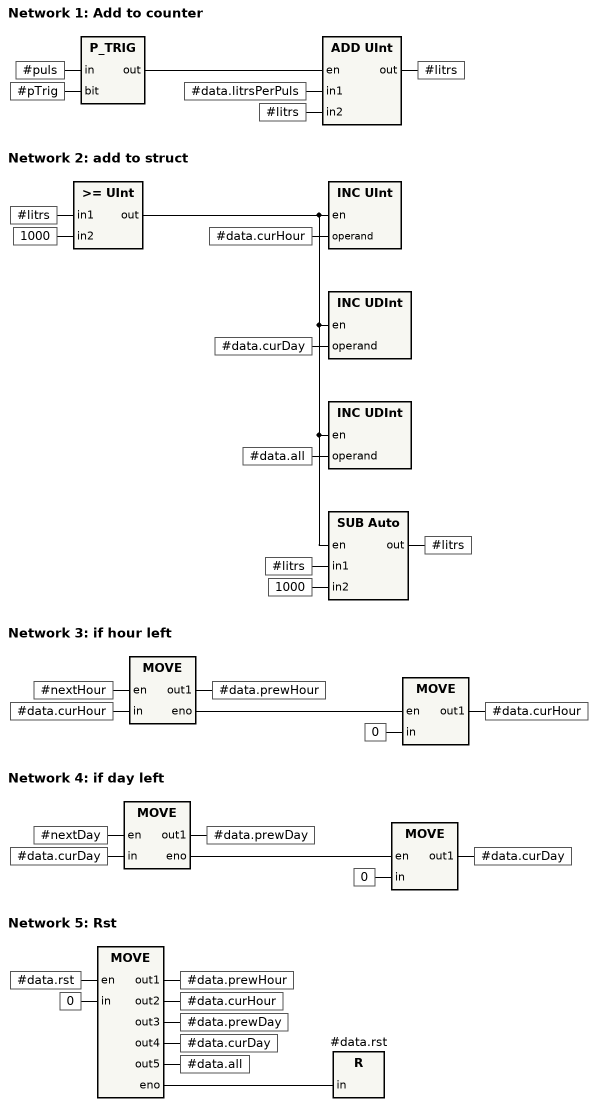
   #_w1 := #puls AND NOT #pTrig;   // rising edge
   #pTrig := #puls;
   IF #_w1 THEN #litrs := #data.litrsPerPuls + #litrs; END_IF;
END_REGION

REGION Network 2: add to struct
   IF #litrs >= 1000 THEN
       #data.curHour := #data.curHour + 1;
       #data.curDay := #data.curDay + 1;
       #data.all := #data.all + 1;
       #litrs := #litrs - 1000;
   END_IF;
END_REGION

REGION Network 3: if hour left
   IF #nextHour THEN
       #data.prewHour := #data.curHour;
       #data.curHour := 0;
   END_IF;
END_REGION

REGION Network 4: if day left
   IF #nextDay THEN
       #data.prewDay := #data.curDay;
       #data.curDay := 0;
   END_IF;
END_REGION

REGION Network 5: Rst
   IF #data.rst THEN
       #data.prewHour := 0;
       #data.curHour := 0;
       #data.prewDay := 0;
       #data.curDay := 0;
       #data.all := 0;
       #data.rst := FALSE;
   END_IF;
END_REGION
END_FUNCTION_BLOCK

FUNCTION "WordToBits" : Void
{ S7_Optimized_Access := 'FALSE' }
VERSION : 0.1
   VAR_INPUT 
      Dev : Word;
   END_VAR

   VAR_OUTPUT 
      Dev1 : Bool;
      Dev2 : Bool;
      Dev3 : Bool;
      Dev4 : Bool;
      Dev5 : Bool;
      Dev6 : Bool;
      Dev7 : Bool;
      Dev8 : Bool;
      Dev9 : Bool;
      Dev10 : Bool;
      Dev11 : Bool;
      Dev12 : Bool;
      Dev13 : Bool;
      Dev14 : Bool;
      Dev15 : Bool;
      Dev16 : Bool;
   END_VAR

   VAR_TEMP 
      TempDev : Word;
      DevBits AT TempDev : Array[1..16] of Bool;
   END_VAR


BEGIN
	#TempDev := #Dev;
	#Dev1 := #DevBits[9];
	#Dev2 := #DevBits[10];
	#Dev3 := #DevBits[11];
	#Dev4 := #DevBits[12];
	#Dev5 := #DevBits[13];
	#Dev6 := #DevBits[14];
	#Dev7 := #DevBits[15];
	#Dev8 := #DevBits[16];
	#Dev9 := #DevBits[1];
	#Dev10 := #DevBits[2];
	#Dev11 := #DevBits[3];
	#Dev12 := #DevBits[4];
	#Dev13 := #DevBits[5];
	#Dev14 := #DevBits[6];
	#Dev15 := #DevBits[7];
	#Dev16 := #DevBits[8];
	
END_FUNCTION

DATA_BLOCK "AllAv_DB"   // DB3
VERSION : 0.1
// stored: AutoNumber true, DBAccessibleFromOPCUA true, InstanceOfName AllAv, InstanceOfType FB
"AllAv"
BEGIN
END_DATA_BLOCK

DATA_BLOCK "AllDpump_DB"   // DB15
VERSION : 0.1
// stored: AutoNumber true, DBAccessibleFromOPCUA true, InstanceOfName AllDpump, InstanceOfType FB
"AllDpump"
BEGIN
END_DATA_BLOCK

DATA_BLOCK "AllPID_DB"   // DB11
VERSION : 0.1
// stored: AutoNumber true, DBAccessibleFromOPCUA true, InstanceOfName AllPID, InstanceOfType FB
"AllPID"
BEGIN
END_DATA_BLOCK

